LIN {X 0,Y 469.67,Z 608.611,A -85,B 0,C 180,E1 -7447.57,E2 -7447.57} C_VEL
LIN {X 0,Y 469.047,Z 617.6,A -85,B 0,C 180,E1 -7449.155,E2 -7449.155} C_VEL
LIN {X 0,Y 468.475,Z 624.989,A -85,B 0,C 180,E1 -7450.73,E2 -7450.73} C_VEL
LIN {X 0,Y 468.024,Z 631.788,A -85,B 0,C 180,E1 -7452.524,E2 -7452.524} C_VEL
LIN {X 0,Y 467.689,Z 637.041,A -85,B 0,C 180,E1 -7454.307,E2 -7454.307} C_VEL
LIN {X 0,Y 467.424,Z 640.917,A -85,B 0,C 180,E1 -7456.081,E2 -7456.081} C_VEL
LIN {X 0,Y 467.26,Z 643.569,A -85,B 0,C 180,E1 -7457.867,E2 -7457.867} C_VEL
LIN {X 0,Y 467.199,Z 644.998,A -85,B 0,C 180,E1 -7459.601,E2 -7459.601} C_VEL
LIN {X 0,Y 467.203,Z 645.333,A -85,B 0,C 180,E1 -7461.349,E2 -7461.349} C_VEL
LIN {X 0,Y 467.285,Z 644.567,A -85,B 0,C 180,E1 -7463.09,E2 -7463.09} C_VEL
LIN {X 0,Y 467.339,Z 642.693,A -85,B 0,C 180,E1 -7464.824,E2 -7464.824} C_VEL
LIN {X 0,Y 467.523,Z 639.635,A -85,B 0,C 180,E1 -7466.553,E2 -7466.553} C_VEL
LIN {X 0,Y 467.688,Z 635.408,A -85,B 0,C 180,E1 -7468.278,E2 -7468.278} C_VEL
LIN {X 0,Y 468.03,Z 629.881,A -85,B 0,C 180,E1 -7470,E2 -7470} C_VEL
LIN {X 0,Y 468.557,Z 622.901,A -85,B 0,C 180,E1 -7471.719,E2 -7471.719} C_VEL
LIN {X 0,Y 469.049,Z 615.461,A -85,B 0,C 180,E1 -7473.221,E2 -7473.221} C_VEL
LIN {X 0,Y 469.708,Z 606.525,A -85,B 0,C 180,E1 -7474.721,E2 -7474.721} C_VEL
LIN {X 0,Y 470.4,Z 597.458,A -85,B 0,C 180,E1 -7476.003,E2 -7476.003} C_VEL
LIN {X 0,Y 471.082,Z 586.721,A -85,B 0,C 180,E1 -7477.285,E2 -7477.285} C_VEL
LIN {X 0,Y 471.807,Z 574.946,A -85,B 0,C 180,E1 -7478.459,E2 -7478.459} C_VEL
LIN {X 0,Y 472.642,Z 561.989,A -85,B 0,C 180,E1 -7479.522,E2 -7479.522} C_VEL
LIN {X 0,Y 473.369,Z 547.59,A -85,B 0,C 180,E1 -7480.479,E2 -7480.479} C_VEL
LIN {X 0,Y 473.972,Z 533.272,A -85,B 0,C 180,E1 -7481.223,E2 -7481.223} C_VEL
LIN {X 0,Y 474.382,Z 517.89,A -85,B 0,C 180,E1 -7481.826,E2 -7481.826} C_VEL
LIN {X 0,Y 474.573,Z 502.138,A -85,B 0,C 180,E1 -7482.25,E2 -7482.25} C_VEL
LIN {X 0,Y 475.64,Z 391.415,A -85,B 0,C 180,E1 -7483.988,E2 -7483.988} C_VEL
LIN {X 0,Y 467.72,Z 373.635,A -85,B 0,C 180,E1 -7484.679,E2 -7484.679} C_VEL
LIN {X 0,Y 467.562,Z 372.871,A -85,B 0,C 180,E1 -7484.716,E2 -7484.716} C_VEL
LIN {X 0,Y 467.562,Z 372.866,A -85,B 0,C 180,E1 -7487.495,E2 -7487.495} C_VEL
LIN {X 0,Y 467.593,Z 372.862,A -85,B 0,C 180,E1 -7490.224,E2 -7490.224} C_VEL
LIN {X 0,Y 467.567,Z 372.868,A -85,B 0,C 180,E1 -7493.523,E2 -7493.523} C_VEL
LIN {X 0,Y 467.525,Z 372.875,A -85,B 0,C 180,E1 -7496.806,E2 -7496.806} C_VEL
LIN {X 0,Y 467.509,Z 372.863,A -85,B 0,C 180,E1 -7499.741,E2 -7499.741} C_VEL
LIN {X 0,Y 467.547,Z 372.871,A -85,B 0,C 180,E1 -7502.761,E2 -7502.761} C_VEL
LIN {X 0,Y 467.54,Z 372.867,A -85,B 0,C 180,E1 -7505.89,E2 -7505.89} C_VEL
LIN {X 0,Y 467.528,Z 372.874,A -85,B 0,C 180,E1 -7509.149,E2 -7509.149} C_VEL
LIN {X 0,Y 467.551,Z 372.871,A -85,B 0,C 180,E1 -7511.405,E2 -7511.405} C_VEL
LIN {X 0,Y 467.551,Z 372.87,A -85,B 0,C 180,E1 -7515.05,E2 -7515.05} C_VEL
LIN {X 0,Y 467.556,Z 372.866,A -85,B 0,C 180,E1 -7518.725,E2 -7518.725} C_VEL
LIN {X 0,Y 467.535,Z 372.866,A -85,B 0,C 180,E1 -7521.952,E2 -7521.952} C_VEL
LIN {X 0,Y 467.543,Z 372.873,A -85,B 0,C 180,E1 -7525.165,E2 -7525.165} C_VEL
LIN {X 0,Y 467.535,Z 372.868,A -85,B 0,C 180,E1 -7528.256,E2 -7528.256} C_VEL
LIN {X 0,Y 467.519,Z 372.873,A -85,B 0,C 180,E1 -7531.246,E2 -7531.246} C_VEL
LIN {X 0,Y 467.553,Z 372.865,A -85,B 0,C 180,E1 -7534.405,E2 -7534.405} C_VEL
LIN {X 0,Y 467.564,Z 372.864,A -85,B 0,C 180,E1 -7536.995,E2 -7536.995} C_VEL
LIN {X 0,Y 467.61,Z 372.859,A -85,B 0,C 180,E1 -7539.776,E2 -7539.776} C_VEL
LIN {X 0,Y 467.58,Z 372.86,A -85,B 0,C 180,E1 -7542.505,E2 -7542.505} C_VEL
LIN {X 0,Y 467.586,Z 372.866,A -85,B 0,C 180,E1 -7545.196,E2 -7545.196} C_VEL
LIN {X 0,Y 467.646,Z 372.839,A -85,B 0,C 180,E1 -7547.854,E2 -7547.854} C_VEL
LIN {X 0,Y 467.62,Z 372.849,A -85,B 0,C 180,E1 -7551.356,E2 -7551.356} C_VEL
LIN {X 0,Y 467.691,Z 372.851,A -85,B 0,C 180,E1 -7553.962,E2 -7553.962} C_VEL
LIN {X 0,Y 467.778,Z 372.838,A -85,B 0,C 180,E1 -7557.416,E2 -7557.416} C_VEL
LIN {X 0,Y 467.814,Z 372.835,A -85,B 0,C 180,E1 -7560,E2 -7560} C_VEL
LIN {X 0,Y 467.809,Z 372.831,A -85,B 0,C 180,E1 -7562.583,E2 -7562.583} C_VEL
LIN {X 0,Y 467.681,Z 372.851,A -85,B 0,C 180,E1 -7566.038,E2 -7566.038} C_VEL
LIN {X 0,Y 467.624,Z 372.853,A -85,B 0,C 180,E1 -7568.644,E2 -7568.644} C_VEL
LIN {X 0,Y 467.646,Z 372.855,A -85,B 0,C 180,E1 -7572.146,E2 -7572.146} C_VEL
LIN {X 0,Y 467.602,Z 372.865,A -85,B 0,C 180,E1 -7575.696,E2 -7575.696} C_VEL
LIN {X 0,Y 467.562,Z 372.861,A -85,B 0,C 180,E1 -7578.748,E2 -7578.748} C_VEL
LIN {X 0,Y 467.548,Z 372.869,A -85,B 0,C 180,E1 -7581.261,E2 -7581.261} C_VEL
LIN {X 0,Y 467.541,Z 372.872,A -85,B 0,C 180,E1 -7583.945,E2 -7583.945} C_VEL
LIN {X 0,Y 467.525,Z 372.867,A -85,B 0,C 180,E1 -7586.806,E2 -7586.806} C_VEL
LIN {X 0,Y 467.531,Z 372.874,A -85,B 0,C 180,E1 -7589.74,E2 -7589.74} C_VEL
LIN {X 0,Y 467.564,Z 372.861,A -85,B 0,C 180,E1 -7592.76,E2 -7592.76} C_VEL
LIN {X 0,Y 467.534,Z 372.877,A -85,B 0,C 180,E1 -7595.891,E2 -7595.891} C_VEL
LIN {X 0,Y 467.533,Z 372.864,A -85,B 0,C 180,E1 -7599.149,E2 -7599.149} C_VEL
LIN {X 0,Y 467.551,Z 372.87,A -85,B 0,C 180,E1 -7601.405,E2 -7601.405} C_VEL
LIN {X 0,Y 467.557,Z 372.865,A -85,B 0,C 180,E1 -7605.052,E2 -7605.052} C_VEL
LIN {X 0,Y 467.546,Z 372.859,A -85,B 0,C 180,E1 -7608.728,E2 -7608.728} C_VEL
LIN {X 0,Y 467.534,Z 372.875,A -85,B 0,C 180,E1 -7611.953,E2 -7611.953} C_VEL
LIN {X 0,Y 467.625,Z 373.006,A -85,B 0,C 180,E1 -7615.296,E2 -7615.296} C_VEL
LIN {X 0,Y 472.99,Z 393.471,A -85,B 0,C 180,E1 -7618.068,E2 -7618.068} C_VEL
LIN {X 0,Y 473.845,Z 397.012,A -85,B 0,C 180,E1 -7618.531,E2 -7618.531} C_VEL
LIN {X 0,Y 472.881,Z 418.835,A -85,B 0,C 180,E1 -7621.031,E2 -7621.031} C_VEL
LIN {X 0,Y 471.759,Z 444.502,A -85,B 0,C 180,E1 -7623.93,E2 -7623.93} C_VEL
LIN {X 0,Y 471.04,Z 462.048,A -85,B 0,C 180,E1 -7625.895,E2 -7625.895} C_VEL
LIN {X 0,Y 475.467,Z 492.83,A -85,B 0,C 180,E1 -7626.599,E2 -7626.599} C_VEL
LIN {X 0,Y 473.858,Z 631.608,A -85,B 0,C 180,E1 -7628.75,E2 -7628.75} C_VEL
LIN {X 0,Y 473.273,Z 647.666,A -85,B 0,C 180,E1 -7629.177,E2 -7629.177} C_VEL
LIN {X 0,Y 472.573,Z 661.612,A -85,B 0,C 180,E1 -7629.705,E2 -7629.705} C_VEL
LIN {X 0,Y 471.782,Z 675.9,A -85,B 0,C 180,E1 -7630.417,E2 -7630.417} C_VEL
LIN {X 0,Y 470.956,Z 689.732,A -85,B 0,C 180,E1 -7631.286,E2 -7631.286} C_VEL
LIN {X 0,Y 470.13,Z 702.495,A -85,B 0,C 180,E1 -7632.267,E2 -7632.267} C_VEL
LIN {X 0,Y 469.317,Z 715.487,A -85,B 0,C 180,E1 -7633.47,E2 -7633.47} C_VEL
LIN {X 0,Y 468.57,Z 727.313,A -85,B 0,C 180,E1 -7634.783,E2 -7634.783} C_VEL
LIN {X 0,Y 468.028,Z 737.298,A -85,B 0,C 180,E1 -7636.098,E2 -7636.098} C_VEL
LIN {X 0,Y 467.584,Z 746.096,A -85,B 0,C 180,E1 -7637.456,E2 -7637.456} C_VEL
LIN {X 0,Y 467.298,Z 754.281,A -85,B 0,C 180,E1 -7638.945,E2 -7638.945} C_VEL
LIN {X 0,Y 467.041,Z 761.256,A -85,B 0,C 180,E1 -7640.472,E2 -7640.472} C_VEL
LIN {X 0,Y 466.972,Z 767.735,A -85,B 0,C 180,E1 -7642.215,E2 -7642.215} C_VEL
LIN {X 0,Y 466.958,Z 772.754,A -85,B 0,C 180,E1 -7643.952,E2 -7643.952} C_VEL
LIN {X 0,Y 467.019,Z 776.441,A -85,B 0,C 180,E1 -7645.685,E2 -7645.685} C_VEL
LIN {X 0,Y 466.958,Z 778.848,A -85,B 0,C 180,E1 -7647.412,E2 -7647.412} C_VEL
LIN {X 0,Y 467.025,Z 780.065,A -85,B 0,C 180,E1 -7649.137,E2 -7649.137} C_VEL
LIN {X 0,Y 467.026,Z 780.047,A -85,B 0,C 180,E1 -7650.862,E2 -7650.862} C_VEL
LIN {X 0,Y 466.964,Z 778.797,A -85,B 0,C 180,E1 -7652.587,E2 -7652.587} C_VEL
LIN {X 0,Y 467.04,Z 776.363,A -85,B 0,C 180,E1 -7654.315,E2 -7654.315} C_VEL
LIN {X 0,Y 466.966,Z 772.648,A -85,B 0,C 180,E1 -7656.047,E2 -7656.047} C_VEL
LIN {X 0,Y 466.981,Z 767.598,A -85,B 0,C 180,E1 -7657.784,E2 -7657.784} C_VEL
LIN {X 0,Y 467.071,Z 761.078,A -85,B 0,C 180,E1 -7659.527,E2 -7659.527} C_VEL
LIN {X 0,Y 467.296,Z 754.064,A -85,B 0,C 180,E1 -7661.055,E2 -7661.055} C_VEL
LIN {X 0,Y 467.591,Z 745.859,A -85,B 0,C 180,E1 -7662.543,E2 -7662.543} C_VEL
LIN {X 0,Y 468.026,Z 737.049,A -85,B 0,C 180,E1 -7663.901,E2 -7663.901} C_VEL
LIN {X 0,Y 468.578,Z 727.074,A -85,B 0,C 180,E1 -7665.216,E2 -7665.216} C_VEL
LIN {X 0,Y 469.304,Z 714.794,A -85,B 0,C 180,E1 -7666.58,E2 -7666.58} C_VEL
LIN {X 0,Y 470.115,Z 702.374,A -85,B 0,C 180,E1 -7667.733,E2 -7667.733} C_VEL
LIN {X 0,Y 470.899,Z 689.72,A -85,B 0,C 180,E1 -7668.715,E2 -7668.715} C_VEL
LIN {X 0,Y 471.784,Z 676.095,A -85,B 0,C 180,E1 -7669.582,E2 -7669.582} C_VEL
LIN {X 0,Y 472.598,Z 662.069,A -85,B 0,C 180,E1 -7670.293,E2 -7670.293} C_VEL
LIN {X 0,Y 473.391,Z 646.192,A -85,B 0,C 180,E1 -7670.901,E2 -7670.901} C_VEL
LIN {X 0,Y 473.955,Z 630.96,A -85,B 0,C 180,E1 -7671.302,E2 -7671.302} C_VEL
LIN {X 0,Y 475.444,Z 512.492,A -85,B 0,C 180,E1 -7673.158,E2 -7673.158} C_VEL
LIN {X 0,Y 475.512,Z 491.468,A -85,B 0,C 180,E1 -7673.495,E2 -7673.495} C_VEL
LIN {X 0,Y 471.127,Z 461.112,A -85,B 0,C 180,E1 -7674.248,E2 -7674.248} C_VEL
LIN {X 0,Y 472.502,Z 431.974,A -85,B 0,C 180,E1 -7677.577,E2 -7677.577} C_VEL
LIN {X 0,Y 473.976,Z 403.693,A -85,B 0,C 180,E1 -7680.877,E2 -7680.877} C_VEL
LIN {X 0,Y 474.148,Z 396.929,A -85,B 0,C 180,E1 -7681.691,E2 -7681.691} C_VEL
LIN {X 0,Y 469.857,Z 380.816,A -85,B 0,C 180,E1 -7683.982,E2 -7683.982} C_VEL
LIN {X 0,Y 467.577,Z 372.866,A -85,B 0,C 180,E1 -7685.192,E2 -7685.192} C_VEL
LIN {X 0,Y 467.533,Z 372.874,A -85,B 0,C 180,E1 -7688.587,E2 -7688.587} C_VEL
LIN {X 0,Y 467.552,Z 372.866,A -85,B 0,C 180,E1 -7691.404,E2 -7691.404} C_VEL
LIN {X 0,Y 467.553,Z 372.858,A -85,B 0,C 180,E1 -7694.947,E2 -7694.947} C_VEL
LIN {X 0,Y 467.547,Z 372.868,A -85,B 0,C 180,E1 -7698.594,E2 -7698.594} C_VEL
LIN {X 0,Y 467.529,Z 372.866,A -85,B 0,C 180,E1 -7701.412,E2 -7701.412} C_VEL
LIN {X 0,Y 467.537,Z 372.872,A -85,B 0,C 180,E1 -7704.262,E2 -7704.262} C_VEL
LIN {X 0,Y 467.559,Z 372.866,A -85,B 0,C 180,E1 -7707.323,E2 -7707.323} C_VEL
LIN {X 0,Y 467.536,Z 372.873,A -85,B 0,C 180,E1 -7710.672,E2 -7710.672} C_VEL
LIN {X 0,Y 467.52,Z 372.871,A -85,B 0,C 180,E1 -7713.194,E2 -7713.194} C_VEL
LIN {X 0,Y 467.536,Z 372.871,A -85,B 0,C 180,E1 -7716.055,E2 -7716.055} C_VEL
LIN {X 0,Y 467.571,Z 372.863,A -85,B 0,C 180,E1 -7719.775,E2 -7719.775} C_VEL
LIN {X 0,Y 467.542,Z 372.871,A -85,B 0,C 180,E1 -7722.504,E2 -7722.504} C_VEL
LIN {X 0,Y 467.571,Z 372.864,A -85,B 0,C 180,E1 -7725.196,E2 -7725.196} C_VEL
LIN {X 0,Y 467.641,Z 372.857,A -85,B 0,C 180,E1 -7727.854,E2 -7727.854} C_VEL
LIN {X 0,Y 467.619,Z 372.858,A -85,B 0,C 180,E1 -7731.356,E2 -7731.356} C_VEL
LIN {X 0,Y 467.677,Z 372.848,A -85,B 0,C 180,E1 -7733.962,E2 -7733.962} C_VEL
LIN {X 0,Y 467.805,Z 372.83,A -85,B 0,C 180,E1 -7737.417,E2 -7737.417} C_VEL
LIN {X 0,Y 467.831,Z 372.833,A -85,B 0,C 180,E1 -7740,E2 -7740} C_VEL
LIN {X 0,Y 467.803,Z 372.84,A -85,B 0,C 180,E1 -7742.583,E2 -7742.583} C_VEL
LIN {X 0,Y 467.706,Z 372.84,A -85,B 0,C 180,E1 -7746.038,E2 -7746.038} C_VEL
LIN {X 0,Y 467.646,Z 372.849,A -85,B 0,C 180,E1 -7748.644,E2 -7748.644} C_VEL
LIN {X 0,Y 467.641,Z 372.856,A -85,B 0,C 180,E1 -7752.146,E2 -7752.146} C_VEL
LIN {X 0,Y 467.636,Z 372.85,A -85,B 0,C 180,E1 -7755.885,E2 -7755.885} C_VEL
LIN {X 0,Y 467.609,Z 372.854,A -85,B 0,C 180,E1 -7759.309,E2 -7759.309} C_VEL
LIN {X 0,Y 467.518,Z 372.864,A -85,B 0,C 180,E1 -7762.075,E2 -7762.075} C_VEL
LIN {X 0,Y 467.543,Z 372.87,A -85,B 0,C 180,E1 -7764.891,E2 -7764.891} C_VEL
LIN {X 0,Y 467.535,Z 372.865,A -85,B 0,C 180,E1 -7767.775,E2 -7767.775} C_VEL
LIN {X 0,Y 467.54,Z 372.866,A -85,B 0,C 180,E1 -7771.042,E2 -7771.042} C_VEL
LIN {X 0,Y 467.567,Z 372.867,A -85,B 0,C 180,E1 -7774.241,E2 -7774.241} C_VEL
LIN {X 0,Y 467.538,Z 372.869,A -85,B 0,C 180,E1 -7777.187,E2 -7777.187} C_VEL
LIN {X 0,Y 467.549,Z 372.866,A -85,B 0,C 180,E1 -7780.268,E2 -7780.268} C_VEL
LIN {X 0,Y 467.539,Z 372.863,A -85,B 0,C 180,E1 -7783.747,E2 -7783.747} C_VEL
LIN {X 0,Y 467.54,Z 372.869,A -85,B 0,C 180,E1 -7786.256,E2 -7786.256} C_VEL
LIN {X 0,Y 467.553,Z 372.866,A -85,B 0,C 180,E1 -7789.735,E2 -7789.735} C_VEL
LIN {X 0,Y 467.538,Z 372.871,A -85,B 0,C 180,E1 -7792.816,E2 -7792.816} C_VEL
LIN {X 0,Y 467.572,Z 372.868,A -85,B 0,C 180,E1 -7795.761,E2 -7795.761} C_VEL
LIN {X 0,Y 467.592,Z 372.908,A -85,B 0,C 180,E1 -7797.131,E2 -7797.131} C_VEL
LIN {X 0,Y 468.547,Z 375.634,A -85,B 0,C 180,E1 -7797.236,E2 -7797.236} C_VEL
LIN {X 0,Y 476.262,Z 391.882,A -85,B 0,C 180,E1 -7797.966,E2 -7797.966} C_VEL
LIN {X 0,Y 475.026,Z 501.799,A -85,B 0,C 180,E1 -7799.71,E2 -7799.71} C_VEL
LIN {X 0,Y 475.018,Z 504.372,A -85,B 0,C 180,E1 -7799.763,E2 -7799.763} C_VEL
LIN {X 0,Y 474.664,Z 508.241,A -85,B 0,C 180,E1 -7799.84,E2 -7799.84} C_VEL
LIN {X 0,Y 472.596,Z 515.855,A -85,B 0,C 180,E1 -7799.943,E2 -7799.943} C_VEL
LIN {X 0,Y 468.602,Z 527.997,A -85,B 0,C 180,E1 -7800.171,E2 -7800.171} C_VEL
LIN {X 0,Y 467.913,Z 532.637,A -85,B 0,C 180,E1 -7800.343,E2 -7800.343} C_VEL
LIN {X 0,Y 467.847,Z 534.491,A -85,B 0,C 180,E1 -7800.424,E2 -7800.424} C_VEL
LIN {X 0,Y 467.113,Z 549.49,A -85,B 0,C 180,E1 -7801.22,E2 -7801.22} C_VEL
LIN {X 0,Y 466.385,Z 563.17,A -85,B 0,C 180,E1 -7802.152,E2 -7802.152} C_VEL
LIN {X 0,Y 465.508,Z 576.883,A -85,B 0,C 180,E1 -7803.312,E2 -7803.312} C_VEL
LIN {X 0,Y 464.664,Z 588.188,A -85,B 0,C 180,E1 -7804.466,E2 -7804.466} C_VEL
LIN {X 0,Y 463.782,Z 599.464,A -85,B 0,C 180,E1 -7805.85,E2 -7805.85} C_VEL
LIN {X 0,Y 462.959,Z 608.86,A -85,B 0,C 180,E1 -7807.227,E2 -7807.227} C_VEL
LIN {X 0,Y 462.247,Z 617.984,A -85,B 0,C 180,E1 -7808.833,E2 -7808.833} C_VEL
LIN {X 0,Y 461.623,Z 625.471,A -85,B 0,C 180,E1 -7810.432,E2 -7810.432} C_VEL
LIN {X 0,Y 461.126,Z 632.379,A -85,B 0,C 180,E1 -7812.254,E2 -7812.254} C_VEL
LIN {X 0,Y 460.729,Z 637.73,A -85,B 0,C 180,E1 -7814.064,E2 -7814.064} C_VEL
LIN {X 0,Y 460.459,Z 641.695,A -85,B 0,C 180,E1 -7815.866,E2 -7815.866} C_VEL
LIN {X 0,Y 460.26,Z 644.531,A -85,B 0,C 180,E1 -7817.758,E2 -7817.758} C_VEL
LIN {X 0,Y 460.18,Z 645.952,A -85,B 0,C 180,E1 -7819.441,E2 -7819.441} C_VEL
LIN {X 0,Y 460.192,Z 646.37,A -85,B 0,C 180,E1 -7821.216,E2 -7821.216} C_VEL
LIN {X 0,Y 460.269,Z 645.681,A -85,B 0,C 180,E1 -7822.984,E2 -7822.984} C_VEL
LIN {X 0,Y 460.33,Z 643.853,A -85,B 0,C 180,E1 -7824.745,E2 -7824.745} C_VEL
LIN {X 0,Y 460.485,Z 640.888,A -85,B 0,C 180,E1 -7826.5,E2 -7826.5} C_VEL
LIN {X 0,Y 460.692,Z 636.744,A -85,B 0,C 180,E1 -7828.252,E2 -7828.252} C_VEL
LIN {X 0,Y 461.044,Z 631.311,A -85,B 0,C 180,E1 -7830,E2 -7830} C_VEL
LIN {X 0,Y 461.586,Z 624.434,A -85,B 0,C 180,E1 -7831.745,E2 -7831.745} C_VEL
LIN {X 0,Y 462.11,Z 617.103,A -85,B 0,C 180,E1 -7833.27,E2 -7833.27} C_VEL
LIN {X 0,Y 462.788,Z 608.296,A -85,B 0,C 180,E1 -7834.791,E2 -7834.791} C_VEL
LIN {X 0,Y 463.52,Z 599.322,A -85,B 0,C 180,E1 -7836.093,E2 -7836.093} C_VEL
LIN {X 0,Y 464.225,Z 588.721,A -85,B 0,C 180,E1 -7837.394,E2 -7837.394} C_VEL
LIN {X 0,Y 464.964,Z 577.141,A -85,B 0,C 180,E1 -7838.584,E2 -7838.584} C_VEL
LIN {X 0,Y 465.853,Z 564.424,A -85,B 0,C 180,E1 -7839.662,E2 -7839.662} C_VEL
LIN {X 0,Y 466.513,Z 552.091,A -85,B 0,C 180,E1 -7840.525,E2 -7840.525} C_VEL
LIN {X 0,Y 467.153,Z 538.751,A -85,B 0,C 180,E1 -7841.278,E2 -7841.278} C_VEL
LIN {X 0,Y 467.643,Z 524.035,A -85,B 0,C 180,E1 -7841.923,E2 -7841.923} C_VEL
LIN {X 0,Y 467.888,Z 509.404,A -85,B 0,C 180,E1 -7842.39,E2 -7842.39} C_VEL
LIN {X 0,Y 468.007,Z 493.494,A -85,B 0,C 180,E1 -7842.714,E2 -7842.714} C_VEL
LIN {X 0,Y 469.054,Z 393.357,A -85,B 0,C 180,E1 -7844.288,E2 -7844.288} C_VEL
LIN {X 0,Y 460.595,Z 374.2,A -85,B 0,C 180,E1 -7845.043,E2 -7845.043} C_VEL
LIN {X 0,Y 460.516,Z 373.749,A -85,B 0,C 180,E1 -7845.093,E2 -7845.093} C_VEL
LIN {X 0,Y 460.516,Z 373.744,A -85,B 0,C 180,E1 -7847.771,E2 -7847.771} C_VEL
LIN {X 0,Y 460.527,Z 373.744,A -85,B 0,C 180,E1 -7850.548,E2 -7850.548} C_VEL
LIN {X 0,Y 460.504,Z 373.747,A -85,B 0,C 180,E1 -7853.695,E2 -7853.695} C_VEL
LIN {X 0,Y 460.479,Z 373.749,A -85,B 0,C 180,E1 -7856.27,E2 -7856.27} C_VEL
LIN {X 0,Y 460.497,Z 373.741,A -85,B 0,C 180,E1 -7859.233,E2 -7859.233} C_VEL
LIN {X 0,Y 460.496,Z 373.746,A -85,B 0,C 180,E1 -7862.287,E2 -7862.287} C_VEL
LIN {X 0,Y 460.496,Z 373.749,A -85,B 0,C 180,E1 -7865.446,E2 -7865.446} C_VEL
LIN {X 0,Y 460.481,Z 373.752,A -85,B 0,C 180,E1 -7868.887,E2 -7868.887} C_VEL
LIN {X 0,Y 460.496,Z 373.748,A -85,B 0,C 180,E1 -7871.597,E2 -7871.597} C_VEL
LIN {X 0,Y 460.494,Z 373.744,A -85,B 0,C 180,E1 -7874.59,E2 -7874.59} C_VEL
LIN {X 0,Y 460.469,Z 373.748,A -85,B 0,C 180,E1 -7877.812,E2 -7877.812} C_VEL
LIN {X 0,Y 460.504,Z 373.744,A -85,B 0,C 180,E1 -7880.134,E2 -7880.134} C_VEL
LIN {X 0,Y 460.458,Z 373.756,A -85,B 0,C 180,E1 -7883.469,E2 -7883.469} C_VEL
LIN {X 0,Y 460.494,Z 373.742,A -85,B 0,C 180,E1 -7886.672,E2 -7886.672} C_VEL
LIN {X 0,Y 460.472,Z 373.748,A -85,B 0,C 180,E1 -7889.757,E2 -7889.757} C_VEL
LIN {X 0,Y 460.476,Z 373.748,A -85,B 0,C 180,E1 -7892.75,E2 -7892.75} C_VEL
LIN {X 0,Y 460.504,Z 373.743,A -85,B 0,C 180,E1 -7895.665,E2 -7895.665} C_VEL
LIN {X 0,Y 460.514,Z 373.743,A -85,B 0,C 180,E1 -7898.578,E2 -7898.578} C_VEL
LIN {X 0,Y 460.574,Z 373.736,A -85,B 0,C 180,E1 -7901.31,E2 -7901.31} C_VEL
LIN {X 0,Y 460.578,Z 373.735,A -85,B 0,C 180,E1 -7904.058,E2 -7904.058} C_VEL
LIN {X 0,Y 460.6,Z 373.718,A -85,B 0,C 180,E1 -7907.665,E2 -7907.665} C_VEL
LIN {X 0,Y 460.576,Z 373.724,A -85,B 0,C 180,E1 -7911.223,E2 -7911.223} C_VEL
LIN {X 0,Y 460.657,Z 373.728,A -85,B 0,C 180,E1 -7913.869,E2 -7913.869} C_VEL
LIN {X 0,Y 460.725,Z 373.716,A -85,B 0,C 180,E1 -7917.377,E2 -7917.377} C_VEL
LIN {X 0,Y 460.764,Z 373.713,A -85,B 0,C 180,E1 -7920,E2 -7920} C_VEL
LIN {X 0,Y 460.753,Z 373.71,A -85,B 0,C 180,E1 -7922.623,E2 -7922.623} C_VEL
LIN {X 0,Y 460.648,Z 373.727,A -85,B 0,C 180,E1 -7926.131,E2 -7926.131} C_VEL
LIN {X 0,Y 460.579,Z 373.73,A -85,B 0,C 180,E1 -7928.777,E2 -7928.777} C_VEL
LIN {X 0,Y 460.599,Z 373.732,A -85,B 0,C 180,E1 -7932.334,E2 -7932.334} C_VEL
LIN {X 0,Y 460.548,Z 373.743,A -85,B 0,C 180,E1 -7935.978,E2 -7935.978} C_VEL
LIN {X 0,Y 460.52,Z 373.738,A -85,B 0,C 180,E1 -7938.886,E2 -7938.886} C_VEL
LIN {X 0,Y 460.499,Z 373.75,A -85,B 0,C 180,E1 -7941.486,E2 -7941.486} C_VEL
LIN {X 0,Y 460.506,Z 373.745,A -85,B 0,C 180,E1 -7944.334,E2 -7944.334} C_VEL
LIN {X 0,Y 460.481,Z 373.747,A -85,B 0,C 180,E1 -7947.249,E2 -7947.249} C_VEL
LIN {X 0,Y 460.492,Z 373.749,A -85,B 0,C 180,E1 -7950.241,E2 -7950.241} C_VEL
LIN {X 0,Y 460.507,Z 373.743,A -85,B 0,C 180,E1 -7953.326,E2 -7953.326} C_VEL
LIN {X 0,Y 460.451,Z 373.753,A -85,B 0,C 180,E1 -7956.532,E2 -7956.532} C_VEL
LIN {X 0,Y 460.501,Z 373.749,A -85,B 0,C 180,E1 -7959.865,E2 -7959.865} C_VEL
LIN {X 0,Y 460.452,Z 373.748,A -85,B 0,C 180,E1 -7962.893,E2 -7962.893} C_VEL
LIN {X 0,Y 460.497,Z 373.747,A -85,B 0,C 180,E1 -7965.832,E2 -7965.832} C_VEL
LIN {X 0,Y 460.495,Z 373.736,A -85,B 0,C 180,E1 -7968.986,E2 -7968.986} C_VEL
LIN {X 0,Y 460.477,Z 373.753,A -85,B 0,C 180,E1 -7972.375,E2 -7972.375} C_VEL
LIN {X 0,Y 460.537,Z 373.758,A -85,B 0,C 180,E1 -7974.956,E2 -7974.956} C_VEL
LIN {X 0,Y 465.718,Z 393.481,A -85,B 0,C 180,E1 -7977.68,E2 -7977.68} C_VEL
LIN {X 0,Y 467.055,Z 399.5,A -85,B 0,C 180,E1 -7978.474,E2 -7978.474} C_VEL
LIN {X 0,Y 465.927,Z 422.481,A -85,B 0,C 180,E1 -7981.14,E2 -7981.14} C_VEL
LIN {X 0,Y 464.771,Z 447.384,A -85,B 0,C 180,E1 -7983.991,E2 -7983.991} C_VEL
LIN {X 0,Y 464.175,Z 461.003,A -85,B 0,C 180,E1 -7985.539,E2 -7985.539} C_VEL
LIN {X 0,Y 468.822,Z 493.715,A -85,B 0,C 180,E1 -7986.299,E2 -7986.299} C_VEL
LIN {X 0,Y 467.199,Z 629.756,A -85,B 0,C 180,E1 -7988.432,E2 -7988.432} C_VEL
LIN {X 0,Y 466.625,Z 645.698,A -85,B 0,C 180,E1 -7988.85,E2 -7988.85} C_VEL
LIN {X 0,Y 465.829,Z 660.502,A -85,B 0,C 180,E1 -7989.411,E2 -7989.411} C_VEL
LIN {X 0,Y 465.022,Z 674.608,A -85,B 0,C 180,E1 -7990.12,E2 -7990.12} C_VEL
LIN {X 0,Y 464.097,Z 688.498,A -85,B 0,C 180,E1 -7990.999,E2 -7990.999} C_VEL
LIN {X 0,Y 463.256,Z 701.315,A -85,B 0,C 180,E1 -7991.995,E2 -7991.995} C_VEL
LIN {X 0,Y 462.473,Z 713.255,A -85,B 0,C 180,E1 -7993.104,E2 -7993.104} C_VEL
LIN {X 0,Y 461.714,Z 724.368,A -85,B 0,C 180,E1 -7994.325,E2 -7994.325} C_VEL
LIN {X 0,Y 461.078,Z 734.675,A -85,B 0,C 180,E1 -7995.659,E2 -7995.659} C_VEL
LIN {X 0,Y 460.573,Z 744.783,A -85,B 0,C 180,E1 -7997.217,E2 -7997.217} C_VEL
LIN {X 0,Y 460.226,Z 753.234,A -85,B 0,C 180,E1 -7998.773,E2 -7998.773} C_VEL
LIN {X 0,Y 459.97,Z 760.223,A -85,B 0,C 180,E1 -8000.324,E2 -8000.324} C_VEL
LIN {X 0,Y 459.93,Z 766.715,A -85,B 0,C 180,E1 -8002.095,E2 -8002.095} C_VEL
LIN {X 0,Y 459.907,Z 771.737,A -85,B 0,C 180,E1 -8003.859,E2 -8003.859} C_VEL
LIN {X 0,Y 459.974,Z 775.427,A -85,B 0,C 180,E1 -8005.618,E2 -8005.618} C_VEL
LIN {X 0,Y 459.92,Z 777.835,A -85,B 0,C 180,E1 -8007.372,E2 -8007.372} C_VEL
LIN {X 0,Y 460.011,Z 779.054,A -85,B 0,C 180,E1 -8009.124,E2 -8009.124} C_VEL
LIN {X 0,Y 460.011,Z 779.033,A -85,B 0,C 180,E1 -8010.875,E2 -8010.875} C_VEL
LIN {X 0,Y 459.926,Z 777.776,A -85,B 0,C 180,E1 -8012.627,E2 -8012.627} C_VEL
LIN {X 0,Y 459.996,Z 775.336,A -85,B 0,C 180,E1 -8014.381,E2 -8014.381} C_VEL
LIN {X 0,Y 459.918,Z 771.617,A -85,B 0,C 180,E1 -8016.14,E2 -8016.14} C_VEL
LIN {X 0,Y 459.936,Z 766.563,A -85,B 0,C 180,E1 -8017.904,E2 -8017.904} C_VEL
LIN {X 0,Y 459.991,Z 760.039,A -85,B 0,C 180,E1 -8019.675,E2 -8019.675} C_VEL
LIN {X 0,Y 460.22,Z 753.027,A -85,B 0,C 180,E1 -8021.227,E2 -8021.227} C_VEL
LIN {X 0,Y 460.574,Z 744.583,A -85,B 0,C 180,E1 -8022.782,E2 -8022.782} C_VEL
LIN {X 0,Y 461.098,Z 734.509,A -85,B 0,C 180,E1 -8024.34,E2 -8024.34} C_VEL
LIN {X 0,Y 461.707,Z 724.259,A -85,B 0,C 180,E1 -8025.675,E2 -8025.675} C_VEL
LIN {X 0,Y 462.531,Z 712.158,A -85,B 0,C 180,E1 -8027.007,E2 -8027.007} C_VEL
LIN {X 0,Y 463.445,Z 698.843,A -85,B 0,C 180,E1 -8028.225,E2 -8028.225} C_VEL
LIN {X 0,Y 464.292,Z 685.673,A -85,B 0,C 180,E1 -8029.221,E2 -8029.221} C_VEL
LIN {X 0,Y 465.283,Z 671.331,A -85,B 0,C 180,E1 -8030.098,E2 -8030.098} C_VEL
LIN {X 0,Y 466.169,Z 656.601,A -85,B 0,C 180,E1 -8030.803,E2 -8030.803} C_VEL
LIN {X 0,Y 466.958,Z 641.178,A -85,B 0,C 180,E1 -8031.347,E2 -8031.347} C_VEL
LIN {X 0,Y 467.494,Z 625.052,A -85,B 0,C 180,E1 -8031.727,E2 -8031.727} C_VEL
LIN {X 0,Y 469.125,Z 493.023,A -85,B 0,C 180,E1 -8033.815,E2 -8033.815} C_VEL
LIN {X 0,Y 464.332,Z 459.981,A -85,B 0,C 180,E1 -8034.657,E2 -8034.657} C_VEL
LIN {X 0,Y 465.808,Z 431.181,A -85,B 0,C 180,E1 -8038.008,E2 -8038.008} C_VEL
LIN {X 0,Y 467.299,Z 404.913,A -85,B 0,C 180,E1 -8041.126,E2 -8041.126} C_VEL
LIN {X 0,Y 467.523,Z 399.827,A -85,B 0,C 180,E1 -8041.743,E2 -8041.743} C_VEL
LIN {X 0,Y 464.244,Z 386.595,A -85,B 0,C 180,E1 -8043.631,E2 -8043.631} C_VEL
LIN {X 0,Y 460.521,Z 373.743,A -85,B 0,C 180,E1 -8045.601,E2 -8045.601} C_VEL
LIN {X 0,Y 460.483,Z 373.751,A -85,B 0,C 180,E1 -8048.888,E2 -8048.888} C_VEL
LIN {X 0,Y 460.496,Z 373.747,A -85,B 0,C 180,E1 -8051.598,E2 -8051.598} C_VEL
LIN {X 0,Y 460.501,Z 373.739,A -85,B 0,C 180,E1 -8054.589,E2 -8054.589} C_VEL
LIN {X 0,Y 460.463,Z 373.752,A -85,B 0,C 180,E1 -8057.812,E2 -8057.812} C_VEL
LIN {X 0,Y 460.499,Z 373.751,A -85,B 0,C 180,E1 -8060.134,E2 -8060.134} C_VEL
LIN {X 0,Y 460.447,Z 373.751,A -85,B 0,C 180,E1 -8063.468,E2 -8063.468} C_VEL
LIN {X 0,Y 460.503,Z 373.747,A -85,B 0,C 180,E1 -8066.673,E2 -8066.673} C_VEL
LIN {X 0,Y 460.488,Z 373.746,A -85,B 0,C 180,E1 -8069.759,E2 -8069.759} C_VEL
LIN {X 0,Y 460.477,Z 373.751,A -85,B 0,C 180,E1 -8072.75,E2 -8072.75} C_VEL
LIN {X 0,Y 460.501,Z 373.745,A -85,B 0,C 180,E1 -8075.666,E2 -8075.666} C_VEL
LIN {X 0,Y 460.499,Z 373.747,A -85,B 0,C 180,E1 -8078.581,E2 -8078.581} C_VEL
LIN {X 0,Y 460.515,Z 373.744,A -85,B 0,C 180,E1 -8081.308,E2 -8081.308} C_VEL
LIN {X 0,Y 460.552,Z 373.741,A -85,B 0,C 180,E1 -8084.057,E2 -8084.057} C_VEL
LIN {X 0,Y 460.594,Z 373.733,A -85,B 0,C 180,E1 -8087.666,E2 -8087.666} C_VEL
LIN {X 0,Y 460.574,Z 373.736,A -85,B 0,C 180,E1 -8091.223,E2 -8091.223} C_VEL
LIN {X 0,Y 460.644,Z 373.723,A -85,B 0,C 180,E1 -8093.869,E2 -8093.869} C_VEL
LIN {X 0,Y 460.75,Z 373.709,A -85,B 0,C 180,E1 -8097.377,E2 -8097.377} C_VEL
LIN {X 0,Y 460.78,Z 373.711,A -85,B 0,C 180,E1 -8100,E2 -8100} C_VEL
LIN {X 0,Y 460.747,Z 373.719,A -85,B 0,C 180,E1 -8102.623,E2 -8102.623} C_VEL
LIN {X 0,Y 460.672,Z 373.715,A -85,B 0,C 180,E1 -8106.131,E2 -8106.131} C_VEL
LIN {X 0,Y 460.594,Z 373.729,A -85,B 0,C 180,E1 -8108.777,E2 -8108.777} C_VEL
LIN {X 0,Y 460.595,Z 373.735,A -85,B 0,C 180,E1 -8112.335,E2 -8112.335} C_VEL
LIN {X 0,Y 460.588,Z 373.728,A -85,B 0,C 180,E1 -8115.998,E2 -8115.998} C_VEL
LIN {X 0,Y 460.555,Z 373.731,A -85,B 0,C 180,E1 -8119.616,E2 -8119.616} C_VEL
LIN {X 0,Y 460.495,Z 373.741,A -85,B 0,C 180,E1 -8122.43,E2 -8122.43} C_VEL
LIN {X 0,Y 460.521,Z 373.737,A -85,B 0,C 180,E1 -8125.793,E2 -8125.793} C_VEL
LIN {X 0,Y 460.511,Z 373.748,A -85,B 0,C 180,E1 -8129.233,E2 -8129.233} C_VEL
LIN {X 0,Y 460.515,Z 373.736,A -85,B 0,C 180,E1 -8132.286,E2 -8132.286} C_VEL
LIN {X 0,Y 460.499,Z 373.745,A -85,B 0,C 180,E1 -8135.447,E2 -8135.447} C_VEL
LIN {X 0,Y 460.521,Z 373.75,A -85,B 0,C 180,E1 -8138.896,E2 -8138.896} C_VEL
LIN {X 0,Y 460.471,Z 373.749,A -85,B 0,C 180,E1 -8142.188,E2 -8142.188} C_VEL
LIN {X 0,Y 460.505,Z 373.748,A -85,B 0,C 180,E1 -8145.412,E2 -8145.412} C_VEL
LIN {X 0,Y 460.513,Z 373.747,A -85,B 0,C 180,E1 -8148.988,E2 -8148.988} C_VEL
LIN {X 0,Y 460.509,Z 373.747,A -85,B 0,C 180,E1 -8151.267,E2 -8151.267} C_VEL
LIN {X 0,Y 460.502,Z 373.745,A -85,B 0,C 180,E1 -8154.555,E2 -8154.555} C_VEL
LIN {X 0,Y 460.527,Z 373.746,A -85,B 0,C 180,E1 -8156.676,E2 -8156.676} C_VEL
LIN {X 0,Y 461.674,Z 376.815,A -85,B 0,C 180,E1 -8156.823,E2 -8156.823} C_VEL
LIN {X 0,Y 469.854,Z 393.695,A -85,B 0,C 180,E1 -8157.618,E2 -8157.618} C_VEL
LIN {X 0,Y 468.547,Z 502.603,A -85,B 0,C 180,E1 -8159.37,E2 -8159.37} C_VEL
LIN {X 0,Y 468.329,Z 517.419,A -85,B 0,C 180,E1 -8159.759,E2 -8159.759} C_VEL
LIN {X 0,Y 467.91,Z 531.431,A -85,B 0,C 180,E1 -8160.288,E2 -8160.288} C_VEL
LIN {X 0,Y 467.847,Z 534.491,A -85,B 0,C 180,E1 -8160.424,E2 -8160.424} C_VEL
LIN {X 0,Y 467.117,Z 540.043,A -85,B 0,C 180,E1 -8160.657,E2 -8160.657} C_VEL
LIN {X 0,Y 463.965,Z 549.047,A -85,B 0,C 180,E1 -8161.002,E2 -8161.002} C_VEL
LIN {X 0,Y 460.736,Z 557.83,A -85,B 0,C 180,E1 -8161.413,E2 -8161.413} C_VEL
LIN {X 0,Y 459.863,Z 562.966,A -85,B 0,C 180,E1 -8161.753,E2 -8161.753} C_VEL
LIN {X 0,Y 459.064,Z 575.115,A -85,B 0,C 180,E1 -8162.763,E2 -8162.763} C_VEL
LIN {X 0,Y 458.159,Z 587.034,A -85,B 0,C 180,E1 -8163.955,E2 -8163.955} C_VEL
LIN {X 0,Y 457.213,Z 598.568,A -85,B 0,C 180,E1 -8165.344,E2 -8165.344} C_VEL
LIN {X 0,Y 456.255,Z 609.112,A -85,B 0,C 180,E1 -8166.873,E2 -8166.873} C_VEL
LIN {X 0,Y 455.472,Z 618.368,A -85,B 0,C 180,E1 -8168.503,E2 -8168.503} C_VEL
LIN {X 0,Y 454.767,Z 625.971,A -85,B 0,C 180,E1 -8170.125,E2 -8170.125} C_VEL
LIN {X 0,Y 454.223,Z 632.982,A -85,B 0,C 180,E1 -8171.975,E2 -8171.975} C_VEL
LIN {X 0,Y 453.814,Z 638.427,A -85,B 0,C 180,E1 -8173.815,E2 -8173.815} C_VEL
LIN {X 0,Y 453.483,Z 642.484,A -85,B 0,C 180,E1 -8175.644,E2 -8175.644} C_VEL
LIN {X 0,Y 453.278,Z 645.485,A -85,B 0,C 180,E1 -8177.637,E2 -8177.637} C_VEL
LIN {X 0,Y 453.167,Z 646.909,A -85,B 0,C 180,E1 -8179.275,E2 -8179.275} C_VEL
LIN {X 0,Y 453.191,Z 647.406,A -85,B 0,C 180,E1 -8181.079,E2 -8181.079} C_VEL
LIN {X 0,Y 453.25,Z 646.739,A -85,B 0,C 180,E1 -8182.921,E2 -8182.921} C_VEL
LIN {X 0,Y 453.321,Z 645.008,A -85,B 0,C 180,E1 -8184.663,E2 -8184.663} C_VEL
LIN {X 0,Y 453.449,Z 642.133,A -85,B 0,C 180,E1 -8186.446,E2 -8186.446} C_VEL
LIN {X 0,Y 453.695,Z 638.07,A -85,B 0,C 180,E1 -8188.225,E2 -8188.225} C_VEL
LIN {X 0,Y 454.053,Z 632.731,A -85,B 0,C 180,E1 -8190,E2 -8190} C_VEL
LIN {X 0,Y 454.609,Z 625.954,A -85,B 0,C 180,E1 -8191.772,E2 -8191.772} C_VEL
LIN {X 0,Y 455.163,Z 618.732,A -85,B 0,C 180,E1 -8193.32,E2 -8193.32} C_VEL
LIN {X 0,Y 455.877,Z 610.034,A -85,B 0,C 180,E1 -8194.864,E2 -8194.864} C_VEL
LIN {X 0,Y 456.75,Z 599.555,A -85,B 0,C 180,E1 -8196.405,E2 -8196.405} C_VEL
LIN {X 0,Y 457.564,Z 587.816,A -85,B 0,C 180,E1 -8197.835,E2 -8197.835} C_VEL
LIN {X 0,Y 458.427,Z 575.847,A -85,B 0,C 180,E1 -8199.041,E2 -8199.041} C_VEL
LIN {X 0,Y 459.313,Z 562.637,A -85,B 0,C 180,E1 -8200.135,E2 -8200.135} C_VEL
LIN {X 0,Y 460.008,Z 549.711,A -85,B 0,C 180,E1 -8201.01,E2 -8201.01} C_VEL
LIN {X 0,Y 460.671,Z 535.242,A -85,B 0,C 180,E1 -8201.783,E2 -8201.783} C_VEL
LIN {X 0,Y 461.134,Z 519.549,A -85,B 0,C 180,E1 -8202.411,E2 -8202.411} C_VEL
LIN {X 0,Y 461.355,Z 504.532,A -85,B 0,C 180,E1 -8202.829,E2 -8202.829} C_VEL
LIN {X 0,Y 462.18,Z 427.238,A -85,B 0,C 180,E1 -8204.081,E2 -8204.081} C_VEL
LIN {X 0,Y 462.518,Z 395.306,A -85,B 0,C 180,E1 -8204.592,E2 -8204.592} C_VEL
LIN {X 0,Y 453.561,Z 375.062,A -85,B 0,C 180,E1 -8205.408,E2 -8205.408} C_VEL
LIN {X 0,Y 453.498,Z 374.621,A -85,B 0,C 180,E1 -8205.426,E2 -8205.426} C_VEL
LIN {X 0,Y 453.487,Z 374.623,A -85,B 0,C 180,E1 -8209.027,E2 -8209.027} C_VEL
LIN {X 0,Y 453.471,Z 374.622,A -85,B 0,C 180,E1 -8211.836,E2 -8211.836} C_VEL
LIN {X 0,Y 453.45,Z 374.628,A -85,B 0,C 180,E1 -8214.738,E2 -8214.738} C_VEL
LIN {X 0,Y 453.456,Z 374.624,A -85,B 0,C 180,E1 -8217.941,E2 -8217.941} C_VEL
LIN {X 0,Y 453.446,Z 374.618,A -85,B 0,C 180,E1 -8220.761,E2 -8220.761} C_VEL
LIN {X 0,Y 453.453,Z 374.621,A -85,B 0,C 180,E1 -8223.914,E2 -8223.914} C_VEL
LIN {X 0,Y 453.432,Z 374.629,A -85,B 0,C 180,E1 -8227.191,E2 -8227.191} C_VEL
LIN {X 0,Y 453.465,Z 374.619,A -85,B 0,C 180,E1 -8230.611,E2 -8230.611} C_VEL
LIN {X 0,Y 453.436,Z 374.622,A -85,B 0,C 180,E1 -8234.224,E2 -8234.224} C_VEL
LIN {X 0,Y 453.411,Z 374.632,A -85,B 0,C 180,E1 -8236.999,E2 -8236.999} C_VEL
LIN {X 0,Y 453.466,Z 374.627,A -85,B 0,C 180,E1 -8239.412,E2 -8239.412} C_VEL
LIN {X 0,Y 453.432,Z 374.625,A -85,B 0,C 180,E1 -8242.808,E2 -8242.808} C_VEL
LIN {X 0,Y 453.449,Z 374.618,A -85,B 0,C 180,E1 -8246.085,E2 -8246.085} C_VEL
LIN {X 0,Y 453.44,Z 374.631,A -85,B 0,C 180,E1 -8249.237,E2 -8249.237} C_VEL
LIN {X 0,Y 453.462,Z 374.62,A -85,B 0,C 180,E1 -8252.292,E2 -8252.292} C_VEL
LIN {X 0,Y 453.454,Z 374.625,A -85,B 0,C 180,E1 -8255.262,E2 -8255.262} C_VEL
LIN {X 0,Y 453.473,Z 374.62,A -85,B 0,C 180,E1 -8258.415,E2 -8258.415} C_VEL
LIN {X 0,Y 453.515,Z 374.615,A -85,B 0,C 180,E1 -8261.008,E2 -8261.008} C_VEL
LIN {X 0,Y 453.53,Z 374.614,A -85,B 0,C 180,E1 -8263.893,E2 -8263.893} C_VEL
LIN {X 0,Y 453.556,Z 374.597,A -85,B 0,C 180,E1 -8267.471,E2 -8267.471} C_VEL
LIN {X 0,Y 453.547,Z 374.597,A -85,B 0,C 180,E1 -8271.085,E2 -8271.085} C_VEL
LIN {X 0,Y 453.625,Z 374.605,A -85,B 0,C 180,E1 -8273.774,E2 -8273.774} C_VEL
LIN {X 0,Y 453.674,Z 374.595,A -85,B 0,C 180,E1 -8277.336,E2 -8277.336} C_VEL
LIN {X 0,Y 453.715,Z 374.591,A -85,B 0,C 180,E1 -8280,E2 -8280} C_VEL
LIN {X 0,Y 453.7,Z 374.588,A -85,B 0,C 180,E1 -8282.663,E2 -8282.663} C_VEL
LIN {X 0,Y 453.616,Z 374.602,A -85,B 0,C 180,E1 -8286.226,E2 -8286.226} C_VEL
LIN {X 0,Y 453.55,Z 374.606,A -85,B 0,C 180,E1 -8288.914,E2 -8288.914} C_VEL
LIN {X 0,Y 453.555,Z 374.609,A -85,B 0,C 180,E1 -8292.529,E2 -8292.529} C_VEL
LIN {X 0,Y 453.487,Z 374.62,A -85,B 0,C 180,E1 -8296.198,E2 -8296.198} C_VEL
LIN {X 0,Y 453.476,Z 374.616,A -85,B 0,C 180,E1 -8299.028,E2 -8299.028} C_VEL
LIN {X 0,Y 453.46,Z 374.625,A -85,B 0,C 180,E1 -8301.837,E2 -8301.837} C_VEL
LIN {X 0,Y 453.459,Z 374.622,A -85,B 0,C 180,E1 -8304.737,E2 -8304.737} C_VEL
LIN {X 0,Y 453.453,Z 374.628,A -85,B 0,C 180,E1 -8307.943,E2 -8307.943} C_VEL
LIN {X 0,Y 453.448,Z 374.624,A -85,B 0,C 180,E1 -8310.761,E2 -8310.761} C_VEL
LIN {X 0,Y 453.457,Z 374.619,A -85,B 0,C 180,E1 -8313.914,E2 -8313.914} C_VEL
LIN {X 0,Y 453.427,Z 374.629,A -85,B 0,C 180,E1 -8317.192,E2 -8317.192} C_VEL
LIN {X 0,Y 453.463,Z 374.622,A -85,B 0,C 180,E1 -8320.612,E2 -8320.612} C_VEL
LIN {X 0,Y 453.473,Z 374.621,A -85,B 0,C 180,E1 -8324.528,E2 -8324.528} C_VEL
LIN {X 0,Y 453.426,Z 374.623,A -85,B 0,C 180,E1 -8328.072,E2 -8328.072} C_VEL
LIN {X 0,Y 453.42,Z 374.628,A -85,B 0,C 180,E1 -8330.805,E2 -8330.805} C_VEL
LIN {X 0,Y 453.437,Z 374.628,A -85,B 0,C 180,E1 -8333.916,E2 -8333.916} C_VEL
LIN {X 0,Y 453.492,Z 374.78,A -85,B 0,C 180,E1 -8334.642,E2 -8334.642} C_VEL
LIN {X 0,Y 458.449,Z 393.398,A -85,B 0,C 180,E1 -8337.27,E2 -8337.27} C_VEL
LIN {X 0,Y 460.265,Z 401.344,A -85,B 0,C 180,E1 -8338.34,E2 -8338.34} C_VEL
LIN {X 0,Y 459.036,Z 424.137,A -85,B 0,C 180,E1 -8341.02,E2 -8341.02} C_VEL
LIN {X 0,Y 457.869,Z 448.164,A -85,B 0,C 180,E1 -8343.814,E2 -8343.814} C_VEL
LIN {X 0,Y 457.304,Z 459.841,A -85,B 0,C 180,E1 -8345.162,E2 -8345.162} C_VEL
LIN {X 0,Y 462.211,Z 494.419,A -85,B 0,C 180,E1 -8345.991,E2 -8345.991} C_VEL
LIN {X 0,Y 460.524,Z 629.097,A -85,B 0,C 180,E1 -8348.133,E2 -8348.133} C_VEL
LIN {X 0,Y 459.891,Z 645.072,A -85,B 0,C 180,E1 -8348.56,E2 -8348.56} C_VEL
LIN {X 0,Y 459.124,Z 659.012,A -85,B 0,C 180,E1 -8349.096,E2 -8349.096} C_VEL
LIN {X 0,Y 458.231,Z 673.234,A -85,B 0,C 180,E1 -8349.813,E2 -8349.813} C_VEL
LIN {X 0,Y 457.265,Z 687.207,A -85,B 0,C 180,E1 -8350.704,E2 -8350.704} C_VEL
LIN {X 0,Y 456.381,Z 700.083,A -85,B 0,C 180,E1 -8351.714,E2 -8351.714} C_VEL
LIN {X 0,Y 455.543,Z 712.067,A -85,B 0,C 180,E1 -8352.839,E2 -8352.839} C_VEL
LIN {X 0,Y 454.711,Z 723.213,A -85,B 0,C 180,E1 -8354.077,E2 -8354.077} C_VEL
LIN {X 0,Y 454.063,Z 733.553,A -85,B 0,C 180,E1 -8355.433,E2 -8355.433} C_VEL
LIN {X 0,Y 453.528,Z 743.69,A -85,B 0,C 180,E1 -8357.015,E2 -8357.015} C_VEL
LIN {X 0,Y 453.17,Z 752.163,A -85,B 0,C 180,E1 -8358.595,E2 -8358.595} C_VEL
LIN {X 0,Y 452.914,Z 759.165,A -85,B 0,C 180,E1 -8360.172,E2 -8360.172} C_VEL
LIN {X 0,Y 452.87,Z 765.675,A -85,B 0,C 180,E1 -8361.971,E2 -8361.971} C_VEL
LIN {X 0,Y 452.859,Z 770.71,A -85,B 0,C 180,E1 -8363.763,E2 -8363.763} C_VEL
LIN {X 0,Y 452.93,Z 774.407,A -85,B 0,C 180,E1 -8365.55,E2 -8365.55} C_VEL
LIN {X 0,Y 452.881,Z 776.818,A -85,B 0,C 180,E1 -8367.331,E2 -8367.331} C_VEL
LIN {X 0,Y 452.995,Z 778.042,A -85,B 0,C 180,E1 -8369.111,E2 -8369.111} C_VEL
LIN {X 0,Y 452.995,Z 778.019,A -85,B 0,C 180,E1 -8370.889,E2 -8370.889} C_VEL
LIN {X 0,Y 452.888,Z 776.758,A -85,B 0,C 180,E1 -8372.668,E2 -8372.668} C_VEL
LIN {X 0,Y 452.952,Z 774.316,A -85,B 0,C 180,E1 -8374.449,E2 -8374.449} C_VEL
LIN {X 0,Y 452.875,Z 770.597,A -85,B 0,C 180,E1 -8376.236,E2 -8376.236} C_VEL
LIN {X 0,Y 452.874,Z 765.545,A -85,B 0,C 180,E1 -8378.028,E2 -8378.028} C_VEL
LIN {X 0,Y 452.926,Z 759.028,A -85,B 0,C 180,E1 -8379.827,E2 -8379.827} C_VEL
LIN {X 0,Y 453.159,Z 752.019,A -85,B 0,C 180,E1 -8381.404,E2 -8381.404} C_VEL
LIN {X 0,Y 453.596,Z 742.294,A -85,B 0,C 180,E1 -8383.21,E2 -8383.21} C_VEL
LIN {X 0,Y 454.15,Z 731.98,A -85,B 0,C 180,E1 -8384.793,E2 -8384.793} C_VEL
LIN {X 0,Y 454.997,Z 720.053,A -85,B 0,C 180,E1 -8386.315,E2 -8386.315} C_VEL
LIN {X 0,Y 455.857,Z 707.93,A -85,B 0,C 180,E1 -8387.611,E2 -8387.611} C_VEL
LIN {X 0,Y 456.761,Z 695.357,A -85,B 0,C 180,E1 -8388.734,E2 -8388.734} C_VEL
LIN {X 0,Y 457.75,Z 681.69,A -85,B 0,C 180,E1 -8389.74,E2 -8389.74} C_VEL
LIN {X 0,Y 458.83,Z 666.607,A -85,B 0,C 180,E1 -8390.627,E2 -8390.627} C_VEL
LIN {X 0,Y 459.787,Z 651.176,A -85,B 0,C 180,E1 -8391.32,E2 -8391.32} C_VEL
LIN {X 0,Y 460.567,Z 636.242,A -85,B 0,C 180,E1 -8391.805,E2 -8391.805} C_VEL
LIN {X 0,Y 461.038,Z 620.696,A -85,B 0,C 180,E1 -8392.135,E2 -8392.135} C_VEL
LIN {X 0,Y 462.631,Z 493.767,A -85,B 0,C 180,E1 -8394.168,E2 -8394.168} C_VEL
LIN {X 0,Y 457.581,Z 458.999,A -85,B 0,C 180,E1 -8395.061,E2 -8395.061} C_VEL
LIN {X 0,Y 459.147,Z 430.412,A -85,B 0,C 180,E1 -8398.451,E2 -8398.451} C_VEL
LIN {X 0,Y 460.667,Z 405.198,A -85,B 0,C 180,E1 -8401.5,E2 -8401.5} C_VEL
LIN {X 0,Y 460.749,Z 401.141,A -85,B 0,C 180,E1 -8402.008,E2 -8402.008} C_VEL
LIN {X 0,Y 457.376,Z 388.029,A -85,B 0,C 180,E1 -8403.926,E2 -8403.926} C_VEL
LIN {X 0,Y 453.429,Z 374.622,A -85,B 0,C 180,E1 -8406.041,E2 -8406.041} C_VEL
LIN {X 0,Y 453.433,Z 374.629,A -85,B 0,C 180,E1 -8409.454,E2 -8409.454} C_VEL
LIN {X 0,Y 453.431,Z 374.63,A -85,B 0,C 180,E1 -8411.929,E2 -8411.929} C_VEL
LIN {X 0,Y 453.471,Z 374.61,A -85,B 0,C 180,E1 -8415.471,E2 -8415.471} C_VEL
LIN {X 0,Y 453.459,Z 374.621,A -85,B 0,C 180,E1 -8419.387,E2 -8419.387} C_VEL
LIN {X 0,Y 453.423,Z 374.628,A -85,B 0,C 180,E1 -8422.808,E2 -8422.808} C_VEL
LIN {X 0,Y 453.452,Z 374.627,A -85,B 0,C 180,E1 -8426.085,E2 -8426.085} C_VEL
LIN {X 0,Y 453.443,Z 374.622,A -85,B 0,C 180,E1 -8429.238,E2 -8429.238} C_VEL
LIN {X 0,Y 453.459,Z 374.626,A -85,B 0,C 180,E1 -8432.293,E2 -8432.293} C_VEL
LIN {X 0,Y 453.454,Z 374.622,A -85,B 0,C 180,E1 -8435.262,E2 -8435.262} C_VEL
LIN {X 0,Y 453.462,Z 374.626,A -85,B 0,C 180,E1 -8438.417,E2 -8438.417} C_VEL
LIN {X 0,Y 453.471,Z 374.623,A -85,B 0,C 180,E1 -8441.007,E2 -8441.007} C_VEL
LIN {X 0,Y 453.501,Z 374.62,A -85,B 0,C 180,E1 -8444.725,E2 -8444.725} C_VEL
LIN {X 0,Y 453.541,Z 374.619,A -85,B 0,C 180,E1 -8448.379,E2 -8448.379} C_VEL
LIN {X 0,Y 453.545,Z 374.613,A -85,B 0,C 180,E1 -8451.086,E2 -8451.086} C_VEL
LIN {X 0,Y 453.612,Z 374.599,A -85,B 0,C 180,E1 -8453.774,E2 -8453.774} C_VEL
LIN {X 0,Y 453.697,Z 374.587,A -85,B 0,C 180,E1 -8457.337,E2 -8457.337} C_VEL
LIN {X 0,Y 453.73,Z 374.589,A -85,B 0,C 180,E1 -8460,E2 -8460} C_VEL
LIN {X 0,Y 453.694,Z 374.598,A -85,B 0,C 180,E1 -8462.664,E2 -8462.664} C_VEL
LIN {X 0,Y 453.64,Z 374.589,A -85,B 0,C 180,E1 -8466.226,E2 -8466.226} C_VEL
LIN {X 0,Y 453.56,Z 374.608,A -85,B 0,C 180,E1 -8468.914,E2 -8468.914} C_VEL
LIN {X 0,Y 453.551,Z 374.61,A -85,B 0,C 180,E1 -8472.529,E2 -8472.529} C_VEL
LIN {X 0,Y 453.532,Z 374.608,A -85,B 0,C 180,E1 -8476.197,E2 -8476.197} C_VEL
LIN {X 0,Y 453.504,Z 374.613,A -85,B 0,C 180,E1 -8479.04,E2 -8479.04} C_VEL
LIN {X 0,Y 453.463,Z 374.613,A -85,B 0,C 180,E1 -8481.837,E2 -8481.837} C_VEL
LIN {X 0,Y 453.473,Z 374.625,A -85,B 0,C 180,E1 -8484.737,E2 -8484.737} C_VEL
LIN {X 0,Y 453.452,Z 374.619,A -85,B 0,C 180,E1 -8487.944,E2 -8487.944} C_VEL
LIN {X 0,Y 453.456,Z 374.625,A -85,B 0,C 180,E1 -8490.761,E2 -8490.761} C_VEL
LIN {X 0,Y 453.457,Z 374.624,A -85,B 0,C 180,E1 -8493.915,E2 -8493.915} C_VEL
LIN {X 0,Y 453.443,Z 374.624,A -85,B 0,C 180,E1 -8497.191,E2 -8497.191} C_VEL
LIN {X 0,Y 453.462,Z 374.62,A -85,B 0,C 180,E1 -8500.613,E2 -8500.613} C_VEL
LIN {X 0,Y 453.452,Z 374.617,A -85,B 0,C 180,E1 -8504.223,E2 -8504.223} C_VEL
LIN {X 0,Y 453.431,Z 374.626,A -85,B 0,C 180,E1 -8507.003,E2 -8507.003} C_VEL
LIN {X 0,Y 453.465,Z 374.621,A -85,B 0,C 180,E1 -8509.414,E2 -8509.414} C_VEL
LIN {X 0,Y 453.445,Z 374.626,A -85,B 0,C 180,E1 -8512.811,E2 -8512.811} C_VEL
LIN {X 0,Y 453.482,Z 374.623,A -85,B 0,C 180,E1 -8516.239,E2 -8516.239} C_VEL
LIN {X 0,Y 454.498,Z 377.472,A -85,B 0,C 180,E1 -8516.366,E2 -8516.366} C_VEL
LIN {X 0,Y 463.466,Z 395.727,A -85,B 0,C 180,E1 -8517.261,E2 -8517.261} C_VEL
LIN {X 0,Y 462.1,Z 502.811,A -85,B 0,C 180,E1 -8519.006,E2 -8519.006} C_VEL
LIN {X 0,Y 461.868,Z 518.43,A -85,B 0,C 180,E1 -8519.417,E2 -8519.417} C_VEL
LIN {X 0,Y 461.385,Z 533.53,A -85,B 0,C 180,E1 -8520.002,E2 -8520.002} C_VEL
LIN {X 0,Y 460.725,Z 548.483,A -85,B 0,C 180,E1 -8520.783,E2 -8520.783} C_VEL
LIN {X 0,Y 459.875,Z 562.568,A -85,B 0,C 180,E1 -8521.723,E2 -8521.723} C_VEL
LIN {X 0,Y 459.863,Z 562.966,A -85,B 0,C 180,E1 -8521.753,E2 -8521.753} C_VEL
LIN {X 0,Y 459.014,Z 568.046,A -85,B 0,C 180,E1 -8522.114,E2 -8522.114} C_VEL
LIN {X 0,Y 455.754,Z 576.298,A -85,B 0,C 180,E1 -8522.672,E2 -8522.672} C_VEL
LIN {X 0,Y 452.435,Z 584.277,A -85,B 0,C 180,E1 -8523.29,E2 -8523.29} C_VEL
LIN {X 0,Y 451.464,Z 588.807,A -85,B 0,C 180,E1 -8523.749,E2 -8523.749} C_VEL
LIN {X 0,Y 450.51,Z 599.701,A -85,B 0,C 180,E1 -8525.091,E2 -8525.091} C_VEL
LIN {X 0,Y 449.564,Z 609.385,A -85,B 0,C 180,E1 -8526.508,E2 -8526.508} C_VEL
LIN {X 0,Y 448.706,Z 618.769,A -85,B 0,C 180,E1 -8528.162,E2 -8528.162} C_VEL
LIN {X 0,Y 447.931,Z 626.485,A -85,B 0,C 180,E1 -8529.808,E2 -8529.808} C_VEL
LIN {X 0,Y 447.36,Z 633.594,A -85,B 0,C 180,E1 -8531.688,E2 -8531.688} C_VEL
LIN {X 0,Y 446.87,Z 639.274,A -85,B 0,C 180,E1 -8533.61,E2 -8533.61} C_VEL
LIN {X 0,Y 446.526,Z 643.279,A -85,B 0,C 180,E1 -8535.415,E2 -8535.415} C_VEL
LIN {X 0,Y 446.276,Z 646.462,A -85,B 0,C 180,E1 -8537.525,E2 -8537.525} C_VEL
LIN {X 0,Y 446.156,Z 647.869,A -85,B 0,C 180,E1 -8539.105,E2 -8539.105} C_VEL
LIN {X 0,Y 446.163,Z 648.427,A -85,B 0,C 180,E1 -8540.938,E2 -8540.938} C_VEL
LIN {X 0,Y 446.231,Z 647.788,A -85,B 0,C 180,E1 -8542.856,E2 -8542.856} C_VEL
LIN {X 0,Y 446.312,Z 646.161,A -85,B 0,C 180,E1 -8544.579,E2 -8544.579} C_VEL
LIN {X 0,Y 446.415,Z 643.372,A -85,B 0,C 180,E1 -8546.39,E2 -8546.39} C_VEL
LIN {X 0,Y 446.694,Z 639.389,A -85,B 0,C 180,E1 -8548.197,E2 -8548.197} C_VEL
LIN {X 0,Y 447.057,Z 634.141,A -85,B 0,C 180,E1 -8550,E2 -8550} C_VEL
LIN {X 0,Y 447.645,Z 627.459,A -85,B 0,C 180,E1 -8551.8,E2 -8551.8} C_VEL
LIN {X 0,Y 448.336,Z 619.156,A -85,B 0,C 180,E1 -8553.595,E2 -8553.595} C_VEL
LIN {X 0,Y 449.071,Z 610.352,A -85,B 0,C 180,E1 -8555.163,E2 -8555.163} C_VEL
LIN {X 0,Y 449.864,Z 601.374,A -85,B 0,C 180,E1 -8556.504,E2 -8556.504} C_VEL
LIN {X 0,Y 450.647,Z 590.77,A -85,B 0,C 180,E1 -8557.843,E2 -8557.843} C_VEL
LIN {X 0,Y 451.467,Z 579.185,A -85,B 0,C 180,E1 -8559.069,E2 -8559.069} C_VEL
LIN {X 0,Y 452.429,Z 566.465,A -85,B 0,C 180,E1 -8560.178,E2 -8560.178} C_VEL
LIN {X 0,Y 453.146,Z 554.133,A -85,B 0,C 180,E1 -8561.065,E2 -8561.065} C_VEL
LIN {X 0,Y 453.892,Z 539.701,A -85,B 0,C 180,E1 -8561.896,E2 -8561.896} C_VEL
LIN {X 0,Y 454.401,Z 524.546,A -85,B 0,C 180,E1 -8562.562,E2 -8562.562} C_VEL
LIN {X 0,Y 454.683,Z 509.375,A -85,B 0,C 180,E1 -8563.037,E2 -8563.037} C_VEL
LIN {X 0,Y 454.803,Z 490.439,A -85,B 0,C 180,E1 -8563.403,E2 -8563.403} C_VEL
LIN {X 0,Y 455.964,Z 397.268,A -85,B 0,C 180,E1 -8564.903,E2 -8564.903} C_VEL
LIN {X 0,Y 446.619,Z 376.337,A -85,B 0,C 180,E1 -8565.769,E2 -8565.769} C_VEL
LIN {X 0,Y 446.455,Z 375.497,A -85,B 0,C 180,E1 -8565.83,E2 -8565.83} C_VEL
LIN {X 0,Y 446.434,Z 375.502,A -85,B 0,C 180,E1 -8569.305,E2 -8569.305} C_VEL
LIN {X 0,Y 446.407,Z 375.502,A -85,B 0,C 180,E1 -8572.2,E2 -8572.2} C_VEL
LIN {X 0,Y 446.406,Z 375.507,A -85,B 0,C 180,E1 -8575.155,E2 -8575.155} C_VEL
LIN {X 0,Y 446.415,Z 375.501,A -85,B 0,C 180,E1 -8578.183,E2 -8578.183} C_VEL
LIN {X 0,Y 446.388,Z 375.506,A -85,B 0,C 180,E1 -8581.302,E2 -8581.302} C_VEL
LIN {X 0,Y 446.412,Z 375.499,A -85,B 0,C 180,E1 -8584.524,E2 -8584.524} C_VEL
LIN {X 0,Y 446.386,Z 375.504,A -85,B 0,C 180,E1 -8587.88,E2 -8587.88} C_VEL
LIN {X 0,Y 446.395,Z 375.502,A -85,B 0,C 180,E1 -8590.912,E2 -8590.912} C_VEL
LIN {X 0,Y 446.372,Z 375.503,A -85,B 0,C 180,E1 -8593.849,E2 -8593.849} C_VEL
LIN {X 0,Y 446.375,Z 375.504,A -85,B 0,C 180,E1 -8596.406,E2 -8596.406} C_VEL
LIN {X 0,Y 446.392,Z 375.504,A -85,B 0,C 180,E1 -8599.796,E2 -8599.796} C_VEL
LIN {X 0,Y 446.389,Z 375.508,A -85,B 0,C 180,E1 -8603.253,E2 -8603.253} C_VEL
LIN {X 0,Y 446.419,Z 375.494,A -85,B 0,C 180,E1 -8606.55,E2 -8606.55} C_VEL
LIN {X 0,Y 446.407,Z 375.498,A -85,B 0,C 180,E1 -8609.983,E2 -8609.983} C_VEL
LIN {X 0,Y 446.375,Z 375.505,A -85,B 0,C 180,E1 -8612.832,E2 -8612.832} C_VEL
LIN {X 0,Y 446.415,Z 375.496,A -85,B 0,C 180,E1 -8615.936,E2 -8615.936} C_VEL
LIN {X 0,Y 446.445,Z 375.497,A -85,B 0,C 180,E1 -8618.772,E2 -8618.772} C_VEL
LIN {X 0,Y 446.44,Z 375.498,A -85,B 0,C 180,E1 -8621.648,E2 -8621.648} C_VEL
LIN {X 0,Y 446.468,Z 375.492,A -85,B 0,C 180,E1 -8624.478,E2 -8624.478} C_VEL
LIN {X 0,Y 446.506,Z 375.467,A -85,B 0,C 180,E1 -8628.192,E2 -8628.192} C_VEL
LIN {X 0,Y 446.499,Z 375.473,A -85,B 0,C 180,E1 -8630.944,E2 -8630.944} C_VEL
LIN {X 0,Y 446.595,Z 375.482,A -85,B 0,C 180,E1 -8633.675,E2 -8633.675} C_VEL
LIN {X 0,Y 446.626,Z 375.472,A -85,B 0,C 180,E1 -8637.294,E2 -8637.294} C_VEL
LIN {X 0,Y 446.667,Z 375.469,A -85,B 0,C 180,E1 -8640,E2 -8640} C_VEL
LIN {X 0,Y 446.65,Z 375.466,A -85,B 0,C 180,E1 -8642.705,E2 -8642.705} C_VEL
LIN {X 0,Y 446.589,Z 375.477,A -85,B 0,C 180,E1 -8646.324,E2 -8646.324} C_VEL
LIN {X 0,Y 446.491,Z 375.491,A -85,B 0,C 180,E1 -8649.971,E2 -8649.971} C_VEL
LIN {X 0,Y 446.512,Z 375.486,A -85,B 0,C 180,E1 -8652.73,E2 -8652.73} C_VEL
LIN {X 0,Y 446.441,Z 375.498,A -85,B 0,C 180,E1 -8656.207,E2 -8656.207} C_VEL
LIN {X 0,Y 446.422,Z 375.497,A -85,B 0,C 180,E1 -8659.305,E2 -8659.305} C_VEL
LIN {X 0,Y 446.398,Z 375.5,A -85,B 0,C 180,E1 -8662.2,E2 -8662.2} C_VEL
LIN {X 0,Y 446.412,Z 375.501,A -85,B 0,C 180,E1 -8665.155,E2 -8665.155} C_VEL
LIN {X 0,Y 446.408,Z 375.502,A -85,B 0,C 180,E1 -8668.184,E2 -8668.184} C_VEL
LIN {X 0,Y 446.401,Z 375.504,A -85,B 0,C 180,E1 -8671.301,E2 -8671.301} C_VEL
LIN {X 0,Y 446.412,Z 375.498,A -85,B 0,C 180,E1 -8674.524,E2 -8674.524} C_VEL
LIN {X 0,Y 446.389,Z 375.5,A -85,B 0,C 180,E1 -8678.076,E2 -8678.076} C_VEL
LIN {X 0,Y 446.393,Z 375.506,A -85,B 0,C 180,E1 -8681.395,E2 -8681.395} C_VEL
LIN {X 0,Y 446.414,Z 375.5,A -85,B 0,C 180,E1 -8685.108,E2 -8685.108} C_VEL
LIN {X 0,Y 446.39,Z 375.494,A -85,B 0,C 180,E1 -8688.606,E2 -8688.606} C_VEL
LIN {X 0,Y 446.384,Z 375.509,A -85,B 0,C 180,E1 -8692.12,E2 -8692.12} C_VEL
LIN {X 0,Y 446.449,Z 375.684,A -85,B 0,C 180,E1 -8694.308,E2 -8694.308} C_VEL
LIN {X 0,Y 451.442,Z 394.286,A -85,B 0,C 180,E1 -8696.984,E2 -8696.984} C_VEL
LIN {X 0,Y 453.421,Z 402.154,A -85,B 0,C 180,E1 -8698.073,E2 -8698.073} C_VEL
LIN {X 0,Y 452.373,Z 422.075,A -85,B 0,C 180,E1 -8700.459,E2 -8700.459} C_VEL
LIN {X 0,Y 451.138,Z 445.825,A -85,B 0,C 180,E1 -8703.268,E2 -8703.268} C_VEL
LIN {X 0,Y 450.463,Z 458.974,A -85,B 0,C 180,E1 -8704.809,E2 -8704.809} C_VEL
LIN {X 0,Y 455.577,Z 496.053,A -85,B 0,C 180,E1 -8705.692,E2 -8705.692} C_VEL
LIN {X 0,Y 453.845,Z 628.263,A -85,B 0,C 180,E1 -8707.824,E2 -8707.824} C_VEL
LIN {X 0,Y 453.154,Z 644.379,A -85,B 0,C 180,E1 -8708.263,E2 -8708.263} C_VEL
LIN {X 0,Y 452.306,Z 659.373,A -85,B 0,C 180,E1 -8708.855,E2 -8708.855} C_VEL
LIN {X 0,Y 451.338,Z 673.81,A -85,B 0,C 180,E1 -8709.61,E2 -8709.61} C_VEL
LIN {X 0,Y 450.344,Z 687.482,A -85,B 0,C 180,E1 -8710.514,E2 -8710.514} C_VEL
LIN {X 0,Y 449.338,Z 701.451,A -85,B 0,C 180,E1 -8711.653,E2 -8711.653} C_VEL
LIN {X 0,Y 448.345,Z 714.77,A -85,B 0,C 180,E1 -8712.979,E2 -8712.979} C_VEL
LIN {X 0,Y 447.548,Z 725.719,A -85,B 0,C 180,E1 -8714.283,E2 -8714.283} C_VEL
LIN {X 0,Y 446.809,Z 737.01,A -85,B 0,C 180,E1 -8715.889,E2 -8715.889} C_VEL
LIN {X 0,Y 446.286,Z 746.524,A -85,B 0,C 180,E1 -8717.516,E2 -8717.516} C_VEL
LIN {X 0,Y 446.045,Z 754.233,A -85,B 0,C 180,E1 -8719.101,E2 -8719.101} C_VEL
LIN {X 0,Y 445.811,Z 761.544,A -85,B 0,C 180,E1 -8720.93,E2 -8720.93} C_VEL
LIN {X 0,Y 445.797,Z 767.317,A -85,B 0,C 180,E1 -8722.754,E2 -8722.754} C_VEL
LIN {X 0,Y 445.821,Z 771.682,A -85,B 0,C 180,E1 -8724.572,E2 -8724.572} C_VEL
LIN {X 0,Y 445.837,Z 774.737,A -85,B 0,C 180,E1 -8726.385,E2 -8726.385} C_VEL
LIN {X 0,Y 445.834,Z 776.551,A -85,B 0,C 180,E1 -8728.193,E2 -8728.193} C_VEL
LIN {X 0,Y 445.977,Z 777.028,A -85,B 0,C 180,E1 -8729.097,E2 -8729.097} C_VEL
LIN {X 0,Y 445.978,Z 777.006,A -85,B 0,C 180,E1 -8730.903,E2 -8730.903} C_VEL
LIN {X 0,Y 445.849,Z 775.745,A -85,B 0,C 180,E1 -8732.71,E2 -8732.71} C_VEL
LIN {X 0,Y 445.894,Z 773.304,A -85,B 0,C 180,E1 -8734.52,E2 -8734.52} C_VEL
LIN {X 0,Y 445.834,Z 769.592,A -85,B 0,C 180,E1 -8736.335,E2 -8736.335} C_VEL
LIN {X 0,Y 445.808,Z 764.544,A -85,B 0,C 180,E1 -8738.156,E2 -8738.156} C_VEL
LIN {X 0,Y 445.875,Z 758.038,A -85,B 0,C 180,E1 -8739.984,E2 -8739.984} C_VEL
LIN {X 0,Y 446.103,Z 751.036,A -85,B 0,C 180,E1 -8741.587,E2 -8741.587} C_VEL
LIN {X 0,Y 446.492,Z 742.627,A -85,B 0,C 180,E1 -8743.193,E2 -8743.193} C_VEL
LIN {X 0,Y 447.071,Z 732.599,A -85,B 0,C 180,E1 -8744.8,E2 -8744.8} C_VEL
LIN {X 0,Y 447.773,Z 722.418,A -85,B 0,C 180,E1 -8746.176,E2 -8746.176} C_VEL
LIN {X 0,Y 448.745,Z 710.402,A -85,B 0,C 180,E1 -8747.546,E2 -8747.546} C_VEL
LIN {X 0,Y 449.739,Z 697.195,A -85,B 0,C 180,E1 -8748.801,E2 -8748.801} C_VEL
LIN {X 0,Y 450.753,Z 684.172,A -85,B 0,C 180,E1 -8749.822,E2 -8749.822} C_VEL
LIN {X 0,Y 451.882,Z 670.02,A -85,B 0,C 180,E1 -8750.72,E2 -8750.72} C_VEL
LIN {X 0,Y 452.891,Z 655.035,A -85,B 0,C 180,E1 -8751.467,E2 -8751.467} C_VEL
LIN {X 0,Y 453.783,Z 639.727,A -85,B 0,C 180,E1 -8752.029,E2 -8752.029} C_VEL
LIN {X 0,Y 454.4,Z 624.07,A -85,B 0,C 180,E1 -8752.416,E2 -8752.416} C_VEL
LIN {X 0,Y 456.204,Z 494.77,A -85,B 0,C 180,E1 -8754.526,E2 -8754.526} C_VEL
LIN {X 0,Y 451.296,Z 460.793,A -85,B 0,C 180,E1 -8755.414,E2 -8755.414} C_VEL
LIN {X 0,Y 450.831,Z 457.858,A -85,B 0,C 180,E1 -8755.502,E2 -8755.502} C_VEL
LIN {X 0,Y 452.426,Z 430.668,A -85,B 0,C 180,E1 -8758.786,E2 -8758.786} C_VEL
LIN {X 0,Y 454.007,Z 406.516,A -85,B 0,C 180,E1 -8761.756,E2 -8761.756} C_VEL
LIN {X 0,Y 453.939,Z 402.457,A -85,B 0,C 180,E1 -8762.284,E2 -8762.284} C_VEL
LIN {X 0,Y 449.823,Z 386.804,A -85,B 0,C 180,E1 -8764.64,E2 -8764.64} C_VEL
LIN {X 0,Y 446.393,Z 375.498,A -85,B 0,C 180,E1 -8766.466,E2 -8766.466} C_VEL
LIN {X 0,Y 446.386,Z 375.506,A -85,B 0,C 180,E1 -8769.515,E2 -8769.515} C_VEL
LIN {X 0,Y 446.37,Z 375.506,A -85,B 0,C 180,E1 -8772.61,E2 -8772.61} C_VEL
LIN {X 0,Y 446.411,Z 375.49,A -85,B 0,C 180,E1 -8775.107,E2 -8775.107} C_VEL
LIN {X 0,Y 446.389,Z 375.503,A -85,B 0,C 180,E1 -8778.605,E2 -8778.605} C_VEL
LIN {X 0,Y 446.386,Z 375.504,A -85,B 0,C 180,E1 -8781.923,E2 -8781.923} C_VEL
LIN {X 0,Y 446.407,Z 375.502,A -85,B 0,C 180,E1 -8785.475,E2 -8785.475} C_VEL
LIN {X 0,Y 446.396,Z 375.503,A -85,B 0,C 180,E1 -8788.698,E2 -8788.698} C_VEL
LIN {X 0,Y 446.411,Z 375.504,A -85,B 0,C 180,E1 -8791.836,E2 -8791.836} C_VEL
LIN {X 0,Y 446.407,Z 375.502,A -85,B 0,C 180,E1 -8794.845,E2 -8794.845} C_VEL
LIN {X 0,Y 446.43,Z 375.504,A -85,B 0,C 180,E1 -8798.246,E2 -8798.246} C_VEL
LIN {X 0,Y 446.397,Z 375.503,A -85,B 0,C 180,E1 -8801.647,E2 -8801.647} C_VEL
LIN {X 0,Y 446.442,Z 375.503,A -85,B 0,C 180,E1 -8804.478,E2 -8804.478} C_VEL
LIN {X 0,Y 446.502,Z 375.489,A -85,B 0,C 180,E1 -8807.384,E2 -8807.384} C_VEL
LIN {X 0,Y 446.496,Z 375.492,A -85,B 0,C 180,E1 -8810.944,E2 -8810.944} C_VEL
LIN {X 0,Y 446.583,Z 375.474,A -85,B 0,C 180,E1 -8813.676,E2 -8813.676} C_VEL
LIN {X 0,Y 446.647,Z 375.466,A -85,B 0,C 180,E1 -8817.295,E2 -8817.295} C_VEL
LIN {X 0,Y 446.682,Z 375.467,A -85,B 0,C 180,E1 -8820,E2 -8820} C_VEL
LIN {X 0,Y 446.643,Z 375.477,A -85,B 0,C 180,E1 -8822.706,E2 -8822.706} C_VEL
LIN {X 0,Y 446.609,Z 375.462,A -85,B 0,C 180,E1 -8826.324,E2 -8826.324} C_VEL
LIN {X 0,Y 446.508,Z 375.489,A -85,B 0,C 180,E1 -8829.056,E2 -8829.056} C_VEL
LIN {X 0,Y 446.509,Z 375.483,A -85,B 0,C 180,E1 -8832.73,E2 -8832.73} C_VEL
LIN {X 0,Y 446.476,Z 375.489,A -85,B 0,C 180,E1 -8836.46,E2 -8836.46} C_VEL
LIN {X 0,Y 446.456,Z 375.489,A -85,B 0,C 180,E1 -8839.304,E2 -8839.304} C_VEL
LIN {X 0,Y 446.404,Z 375.494,A -85,B 0,C 180,E1 -8842.201,E2 -8842.201} C_VEL
LIN {X 0,Y 446.417,Z 375.497,A -85,B 0,C 180,E1 -8845.155,E2 -8845.155} C_VEL
LIN {X 0,Y 446.426,Z 375.495,A -85,B 0,C 180,E1 -8848.183,E2 -8848.183} C_VEL
LIN {X 0,Y 446.401,Z 375.495,A -85,B 0,C 180,E1 -8851.302,E2 -8851.302} C_VEL
LIN {X 0,Y 446.413,Z 375.505,A -85,B 0,C 180,E1 -8854.525,E2 -8854.525} C_VEL
LIN {X 0,Y 446.403,Z 375.502,A -85,B 0,C 180,E1 -8858.08,E2 -8858.08} C_VEL
LIN {X 0,Y 446.394,Z 375.505,A -85,B 0,C 180,E1 -8861.395,E2 -8861.395} C_VEL
LIN {X 0,Y 446.443,Z 375.5,A -85,B 0,C 180,E1 -8865.105,E2 -8865.105} C_VEL
LIN {X 0,Y 446.401,Z 375.505,A -85,B 0,C 180,E1 -8868.608,E2 -8868.608} C_VEL
LIN {X 0,Y 446.405,Z 375.498,A -85,B 0,C 180,E1 -8871.923,E2 -8871.923} C_VEL
LIN {X 0,Y 446.42,Z 375.504,A -85,B 0,C 180,E1 -8875.478,E2 -8875.478} C_VEL
LIN {X 0,Y 446.435,Z 375.535,A -85,B 0,C 180,E1 -8875.785,E2 -8875.785} C_VEL
LIN {X 0,Y 447.5,Z 378.441,A -85,B 0,C 180,E1 -8875.91,E2 -8875.91} C_VEL
LIN {X 0,Y 455.892,Z 395.115,A -85,B 0,C 180,E1 -8876.766,E2 -8876.766} C_VEL
LIN {X 0,Y 457.143,Z 397.794,A -85,B 0,C 180,E1 -8876.894,E2 -8876.894} C_VEL
LIN {X 0,Y 455.674,Z 503.937,A -85,B 0,C 180,E1 -8878.649,E2 -8878.649} C_VEL
LIN {X 0,Y 455.431,Z 519.518,A -85,B 0,C 180,E1 -8879.066,E2 -8879.066} C_VEL
LIN {X 0,Y 454.987,Z 533.543,A -85,B 0,C 180,E1 -8879.613,E2 -8879.613} C_VEL
LIN {X 0,Y 454.284,Z 548.517,A -85,B 0,C 180,E1 -8880.392,E2 -8880.392} C_VEL
LIN {X 0,Y 453.468,Z 561.995,A -85,B 0,C 180,E1 -8881.287,E2 -8881.287} C_VEL
LIN {X 0,Y 452.604,Z 574.835,A -85,B 0,C 180,E1 -8882.341,E2 -8882.341} C_VEL
LIN {X 0,Y 451.623,Z 586.979,A -85,B 0,C 180,E1 -8883.549,E2 -8883.549} C_VEL
LIN {X 0,Y 451.464,Z 588.807,A -85,B 0,C 180,E1 -8883.749,E2 -8883.749} C_VEL
LIN {X 0,Y 450.532,Z 593.261,A -85,B 0,C 180,E1 -8884.227,E2 -8884.227} C_VEL
LIN {X 0,Y 447.218,Z 600.463,A -85,B 0,C 180,E1 -8884.987,E2 -8884.987} C_VEL
LIN {X 0,Y 443.81,Z 607.35,A -85,B 0,C 180,E1 -8885.805,E2 -8885.805} C_VEL
LIN {X 0,Y 442.746,Z 611.132,A -85,B 0,C 180,E1 -8886.368,E2 -8886.368} C_VEL
LIN {X 0,Y 441.84,Z 620.408,A -85,B 0,C 180,E1 -8888.051,E2 -8888.051} C_VEL
LIN {X 0,Y 440.976,Z 628.73,A -85,B 0,C 180,E1 -8889.896,E2 -8889.896} C_VEL
LIN {X 0,Y 440.481,Z 634.22,A -85,B 0,C 180,E1 -8891.392,E2 -8891.392} C_VEL
LIN {X 0,Y 439.935,Z 639.854,A -85,B 0,C 180,E1 -8893.289,E2 -8893.289} C_VEL
LIN {X 0,Y 439.555,Z 644.083,A -85,B 0,C 180,E1 -8895.178,E2 -8895.178} C_VEL
LIN {X 0,Y 439.303,Z 647.044,A -85,B 0,C 180,E1 -8897.058,E2 -8897.058} C_VEL
LIN {X 0,Y 439.148,Z 648.827,A -85,B 0,C 180,E1 -8898.929,E2 -8898.929} C_VEL
LIN {X 0,Y 439.149,Z 649.424,A -85,B 0,C 180,E1 -8900.792,E2 -8900.792} C_VEL
LIN {X 0,Y 439.196,Z 648.831,A -85,B 0,C 180,E1 -8902.806,E2 -8902.806} C_VEL
LIN {X 0,Y 439.303,Z 647.31,A -85,B 0,C 180,E1 -8904.492,E2 -8904.492} C_VEL
LIN {X 0,Y 439.381,Z 644.606,A -85,B 0,C 180,E1 -8906.332,E2 -8906.332} C_VEL
LIN {X 0,Y 439.689,Z 640.703,A -85,B 0,C 180,E1 -8908.168,E2 -8908.168} C_VEL
LIN {X 0,Y 440.057,Z 635.542,A -85,B 0,C 180,E1 -8910,E2 -8910} C_VEL
LIN {X 0,Y 440.688,Z 628.945,A -85,B 0,C 180,E1 -8911.828,E2 -8911.828} C_VEL
LIN {X 0,Y 441.387,Z 620.757,A -85,B 0,C 180,E1 -8913.652,E2 -8913.652} C_VEL
LIN {X 0,Y 442.167,Z 612.054,A -85,B 0,C 180,E1 -8915.244,E2 -8915.244} C_VEL
LIN {X 0,Y 443.11,Z 601.572,A -85,B 0,C 180,E1 -8916.832,E2 -8916.832} C_VEL
LIN {X 0,Y 444.042,Z 589.815,A -85,B 0,C 180,E1 -8918.304,E2 -8918.304} C_VEL
LIN {X 0,Y 444.826,Z 579.038,A -85,B 0,C 180,E1 -8919.435,E2 -8919.435} C_VEL
LIN {X 0,Y 445.809,Z 566.074,A -85,B 0,C 180,E1 -8920.56,E2 -8920.56} C_VEL
LIN {X 0,Y 446.571,Z 553.397,A -85,B 0,C 180,E1 -8921.46,E2 -8921.46} C_VEL
LIN {X 0,Y 447.342,Z 538.477,A -85,B 0,C 180,E1 -8922.303,E2 -8922.303} C_VEL
LIN {X 0,Y 447.82,Z 523.694,A -85,B 0,C 180,E1 -8922.936,E2 -8922.936} C_VEL
LIN {X 0,Y 448.095,Z 508.478,A -85,B 0,C 180,E1 -8923.395,E2 -8923.395} C_VEL
LIN {X 0,Y 448.298,Z 482.664,A -85,B 0,C 180,E1 -8923.861,E2 -8923.861} C_VEL
LIN {X 0,Y 449.373,Z 398.996,A -85,B 0,C 180,E1 -8925.228,E2 -8925.228} C_VEL
LIN {X 0,Y 439.502,Z 376.881,A -85,B 0,C 180,E1 -8926.165,E2 -8926.165} C_VEL
LIN {X 0,Y 439.422,Z 376.373,A -85,B 0,C 180,E1 -8926.195,E2 -8926.195} C_VEL
LIN {X 0,Y 439.38,Z 376.378,A -85,B 0,C 180,E1 -8929.627,E2 -8929.627} C_VEL
LIN {X 0,Y 439.351,Z 376.383,A -85,B 0,C 180,E1 -8932.576,E2 -8932.576} C_VEL
LIN {X 0,Y 439.35,Z 376.383,A -85,B 0,C 180,E1 -8935.588,E2 -8935.588} C_VEL
LIN {X 0,Y 439.376,Z 376.381,A -85,B 0,C 180,E1 -8938.676,E2 -8938.676} C_VEL
LIN {X 0,Y 439.341,Z 376.382,A -85,B 0,C 180,E1 -8942.024,E2 -8942.024} C_VEL
LIN {X 0,Y 439.383,Z 376.38,A -85,B 0,C 180,E1 -8945.338,E2 -8945.338} C_VEL
LIN {X 0,Y 439.348,Z 376.381,A -85,B 0,C 180,E1 -8948.598,E2 -8948.598} C_VEL
LIN {X 0,Y 439.358,Z 376.384,A -85,B 0,C 180,E1 -8951.252,E2 -8951.252} C_VEL
LIN {X 0,Y 439.364,Z 376.377,A -85,B 0,C 180,E1 -8954.733,E2 -8954.733} C_VEL
LIN {X 0,Y 439.343,Z 376.38,A -85,B 0,C 180,E1 -8957.789,E2 -8957.789} C_VEL
LIN {X 0,Y 439.349,Z 376.381,A -85,B 0,C 180,E1 -8961.401,E2 -8961.401} C_VEL
LIN {X 0,Y 439.385,Z 376.378,A -85,B 0,C 180,E1 -8964.842,E2 -8964.842} C_VEL
LIN {X 0,Y 439.339,Z 376.382,A -85,B 0,C 180,E1 -8968.136,E2 -8968.136} C_VEL
LIN {X 0,Y 439.37,Z 376.378,A -85,B 0,C 180,E1 -8971.323,E2 -8971.323} C_VEL
LIN {X 0,Y 439.346,Z 376.379,A -85,B 0,C 180,E1 -8974.411,E2 -8974.411} C_VEL
LIN {X 0,Y 439.354,Z 376.383,A -85,B 0,C 180,E1 -8977.424,E2 -8977.424} C_VEL
LIN {X 0,Y 439.434,Z 376.366,A -85,B 0,C 180,E1 -8980.663,E2 -8980.663} C_VEL
LIN {X 0,Y 439.436,Z 376.368,A -85,B 0,C 180,E1 -8984.223,E2 -8984.223} C_VEL
LIN {X 0,Y 439.473,Z 376.344,A -85,B 0,C 180,E1 -8988.001,E2 -8988.001} C_VEL
LIN {X 0,Y 439.47,Z 376.359,A -85,B 0,C 180,E1 -8991.725,E2 -8991.725} C_VEL
LIN {X 0,Y 439.585,Z 376.35,A -85,B 0,C 180,E1 -8994.495,E2 -8994.495} C_VEL
LIN {X 0,Y 439.611,Z 376.341,A -85,B 0,C 180,E1 -8998.167,E2 -8998.167} C_VEL
LIN {X 0,Y 439.619,Z 376.347,A -85,B 0,C 180,E1 -9000,E2 -9000} C_VEL
LIN {X 0,Y 439.602,Z 376.344,A -85,B 0,C 180,E1 -9002.749,E2 -9002.749} C_VEL
LIN {X 0,Y 439.543,Z 376.354,A -85,B 0,C 180,E1 -9006.426,E2 -9006.426} C_VEL
LIN {X 0,Y 439.467,Z 376.363,A -85,B 0,C 180,E1 -9009.202,E2 -9009.202} C_VEL
LIN {X 0,Y 439.455,Z 376.366,A -85,B 0,C 180,E1 -9012.938,E2 -9012.938} C_VEL
LIN {X 0,Y 439.387,Z 376.376,A -85,B 0,C 180,E1 -9016.325,E2 -9016.325} C_VEL
LIN {X 0,Y 439.368,Z 376.379,A -85,B 0,C 180,E1 -9019.628,E2 -9019.628} C_VEL
LIN {X 0,Y 439.343,Z 376.377,A -85,B 0,C 180,E1 -9022.576,E2 -9022.576} C_VEL
LIN {X 0,Y 439.358,Z 376.384,A -85,B 0,C 180,E1 -9025.588,E2 -9025.588} C_VEL
LIN {X 0,Y 439.373,Z 376.376,A -85,B 0,C 180,E1 -9028.676,E2 -9028.676} C_VEL
LIN {X 0,Y 439.357,Z 376.38,A -85,B 0,C 180,E1 -9032.029,E2 -9032.029} C_VEL
LIN {X 0,Y 439.379,Z 376.376,A -85,B 0,C 180,E1 -9035.339,E2 -9035.339} C_VEL
LIN {X 0,Y 439.346,Z 376.374,A -85,B 0,C 180,E1 -9038.599,E2 -9038.599} C_VEL
LIN {X 0,Y 439.356,Z 376.381,A -85,B 0,C 180,E1 -9041.253,E2 -9041.253} C_VEL
LIN {X 0,Y 439.368,Z 376.377,A -85,B 0,C 180,E1 -9044.733,E2 -9044.733} C_VEL
LIN {X 0,Y 439.34,Z 376.382,A -85,B 0,C 180,E1 -9047.79,E2 -9047.79} C_VEL
LIN {X 0,Y 439.344,Z 376.383,A -85,B 0,C 180,E1 -9051.402,E2 -9051.402} C_VEL
LIN {X 0,Y 439.385,Z 376.575,A -85,B 0,C 180,E1 -9053.958,E2 -9053.958} C_VEL
LIN {X 0,Y 444.036,Z 393.667,A -85,B 0,C 180,E1 -9056.476,E2 -9056.476} C_VEL
LIN {X 0,Y 446.673,Z 404.577,A -85,B 0,C 180,E1 -9058.009,E2 -9058.009} C_VEL
LIN {X 0,Y 445.257,Z 427.907,A -85,B 0,C 180,E1 -9060.835,E2 -9060.835} C_VEL
LIN {X 0,Y 444.066,Z 449.651,A -85,B 0,C 180,E1 -9063.443,E2 -9063.443} C_VEL
LIN {X 0,Y 443.599,Z 457.896,A -85,B 0,C 180,E1 -9064.425,E2 -9064.425} C_VEL
LIN {X 0,Y 448.971,Z 496.48,A -85,B 0,C 180,E1 -9065.367,E2 -9065.367} C_VEL
LIN {X 0,Y 447.183,Z 627.296,A -85,B 0,C 180,E1 -9067.506,E2 -9067.506} C_VEL
LIN {X 0,Y 446.485,Z 643.436,A -85,B 0,C 180,E1 -9067.953,E2 -9067.953} C_VEL
LIN {X 0,Y 445.604,Z 657.711,A -85,B 0,C 180,E1 -9068.519,E2 -9068.519} C_VEL
LIN {X 0,Y 444.604,Z 672.341,A -85,B 0,C 180,E1 -9069.287,E2 -9069.287} C_VEL
LIN {X 0,Y 443.515,Z 686.092,A -85,B 0,C 180,E1 -9070.202,E2 -9070.202} C_VEL
LIN {X 0,Y 442.532,Z 698.813,A -85,B 0,C 180,E1 -9071.241,E2 -9071.241} C_VEL
LIN {X 0,Y 441.548,Z 711.697,A -85,B 0,C 180,E1 -9072.507,E2 -9072.507} C_VEL
LIN {X 0,Y 440.669,Z 722.661,A -85,B 0,C 180,E1 -9073.794,E2 -9073.794} C_VEL
LIN {X 0,Y 439.945,Z 732.767,A -85,B 0,C 180,E1 -9075.191,E2 -9075.191} C_VEL
LIN {X 0,Y 439.393,Z 742.709,A -85,B 0,C 180,E1 -9076.825,E2 -9076.825} C_VEL
LIN {X 0,Y 439.007,Z 751.008,A -85,B 0,C 180,E1 -9078.457,E2 -9078.457} C_VEL
LIN {X 0,Y 438.816,Z 756.992,A -85,B 0,C 180,E1 -9079.853,E2 -9079.853} C_VEL
LIN {X 0,Y 438.723,Z 763.538,A -85,B 0,C 180,E1 -9081.71,E2 -9081.71} C_VEL
LIN {X 0,Y 438.759,Z 768.615,A -85,B 0,C 180,E1 -9083.562,E2 -9083.562} C_VEL
LIN {X 0,Y 438.817,Z 772.334,A -85,B 0,C 180,E1 -9085.407,E2 -9085.407} C_VEL
LIN {X 0,Y 438.806,Z 774.77,A -85,B 0,C 180,E1 -9087.246,E2 -9087.246} C_VEL
LIN {X 0,Y 438.958,Z 776.013,A -85,B 0,C 180,E1 -9089.082,E2 -9089.082} C_VEL
LIN {X 0,Y 438.959,Z 775.993,A -85,B 0,C 180,E1 -9090.917,E2 -9090.917} C_VEL
LIN {X 0,Y 438.81,Z 774.736,A -85,B 0,C 180,E1 -9092.754,E2 -9092.754} C_VEL
LIN {X 0,Y 438.837,Z 772.299,A -85,B 0,C 180,E1 -9094.592,E2 -9094.592} C_VEL
LIN {X 0,Y 438.794,Z 768.598,A -85,B 0,C 180,E1 -9096.437,E2 -9096.437} C_VEL
LIN {X 0,Y 438.727,Z 763.554,A -85,B 0,C 180,E1 -9098.289,E2 -9098.289} C_VEL
LIN {X 0,Y 438.816,Z 757.064,A -85,B 0,C 180,E1 -9100.146,E2 -9100.146} C_VEL
LIN {X 0,Y 439.04,Z 750.069,A -85,B 0,C 180,E1 -9101.776,E2 -9101.776} C_VEL
LIN {X 0,Y 439.554,Z 740.402,A -85,B 0,C 180,E1 -9103.64,E2 -9103.64} C_VEL
LIN {X 0,Y 440.204,Z 730.151,A -85,B 0,C 180,E1 -9105.273,E2 -9105.273} C_VEL
LIN {X 0,Y 441.163,Z 718.317,A -85,B 0,C 180,E1 -9106.842,E2 -9106.842} C_VEL
LIN {X 0,Y 442.134,Z 706.288,A -85,B 0,C 180,E1 -9108.176,E2 -9108.176} C_VEL
LIN {X 0,Y 443.273,Z 692.433,A -85,B 0,C 180,E1 -9109.447,E2 -9109.447} C_VEL
LIN {X 0,Y 444.449,Z 678.634,A -85,B 0,C 180,E1 -9110.478,E2 -9110.478} C_VEL
LIN {X 0,Y 445.613,Z 664.035,A -85,B 0,C 180,E1 -9111.349,E2 -9111.349} C_VEL
LIN {X 0,Y 446.644,Z 648.828,A -85,B 0,C 180,E1 -9112.047,E2 -9112.047} C_VEL
LIN {X 0,Y 447.575,Z 632.955,A -85,B 0,C 180,E1 -9112.564,E2 -9112.564} C_VEL
LIN {X 0,Y 448.059,Z 618.525,A -85,B 0,C 180,E1 -9112.873,E2 -9112.873} C_VEL
LIN {X 0,Y 449.783,Z 495.88,A -85,B 0,C 180,E1 -9114.896,E2 -9114.896} C_VEL
LIN {X 0,Y 445.095,Z 462.785,A -85,B 0,C 180,E1 -9115.777,E2 -9115.777} C_VEL
LIN {X 0,Y 444.072,Z 456.654,A -85,B 0,C 180,E1 -9115.97,E2 -9115.97} C_VEL
LIN {X 0,Y 445.808,Z 429.934,A -85,B 0,C 180,E1 -9119.254,E2 -9119.254} C_VEL
LIN {X 0,Y 447.414,Z 407.046,A -85,B 0,C 180,E1 -9122.12,E2 -9122.12} C_VEL
LIN {X 0,Y 447.109,Z 404.029,A -85,B 0,C 180,E1 -9122.538,E2 -9122.538} C_VEL
LIN {X 0,Y 443.246,Z 389.252,A -85,B 0,C 180,E1 -9124.805,E2 -9124.805} C_VEL
LIN {X 0,Y 439.327,Z 376.38,A -85,B 0,C 180,E1 -9126.93,E2 -9126.93} C_VEL
LIN {X 0,Y 439.337,Z 376.385,A -85,B 0,C 180,E1 -9129.839,E2 -9129.839} C_VEL
LIN {X 0,Y 439.327,Z 376.383,A -85,B 0,C 180,E1 -9132.619,E2 -9132.619} C_VEL
LIN {X 0,Y 439.365,Z 376.366,A -85,B 0,C 180,E1 -9135.266,E2 -9135.266} C_VEL
LIN {X 0,Y 439.342,Z 376.38,A -85,B 0,C 180,E1 -9139.015,E2 -9139.015} C_VEL
LIN {X 0,Y 439.344,Z 376.378,A -85,B 0,C 180,E1 -9141.61,E2 -9141.61} C_VEL
LIN {X 0,Y 439.379,Z 376.379,A -85,B 0,C 180,E1 -9144.842,E2 -9144.842} C_VEL
LIN {X 0,Y 439.356,Z 376.385,A -85,B 0,C 180,E1 -9148.138,E2 -9148.138} C_VEL
LIN {X 0,Y 439.374,Z 376.379,A -85,B 0,C 180,E1 -9151.609,E2 -9151.609} C_VEL
LIN {X 0,Y 439.353,Z 376.386,A -85,B 0,C 180,E1 -9154.412,E2 -9154.412} C_VEL
LIN {X 0,Y 439.339,Z 376.383,A -85,B 0,C 180,E1 -9157.423,E2 -9157.423} C_VEL
LIN {X 0,Y 439.371,Z 376.383,A -85,B 0,C 180,E1 -9160.684,E2 -9160.684} C_VEL
LIN {X 0,Y 439.401,Z 376.378,A -85,B 0,C 180,E1 -9164.222,E2 -9164.222} C_VEL
LIN {X 0,Y 439.471,Z 376.365,A -85,B 0,C 180,E1 -9167.285,E2 -9167.285} C_VEL
LIN {X 0,Y 439.463,Z 376.37,A -85,B 0,C 180,E1 -9170.798,E2 -9170.798} C_VEL
LIN {X 0,Y 439.535,Z 376.352,A -85,B 0,C 180,E1 -9173.574,E2 -9173.574} C_VEL
LIN {X 0,Y 439.394,Z 376.374,A -85,B 0,C 180,E1 -9175.413,E2 -9175.413} C_VEL
LIN {X 0,Y 439.615,Z 376.344,A -85,B 0,C 180,E1 -9178.168,E2 -9178.168} C_VEL
LIN {X 0,Y 439.581,Z 376.349,A -85,B 0,C 180,E1 -9180.916,E2 -9180.916} C_VEL
LIN {X 0,Y 439.595,Z 376.355,A -85,B 0,C 180,E1 -9182.749,E2 -9182.749} C_VEL
LIN {X 0,Y 439.581,Z 376.336,A -85,B 0,C 180,E1 -9186.426,E2 -9186.426} C_VEL
LIN {X 0,Y 439.472,Z 376.364,A -85,B 0,C 180,E1 -9189.202,E2 -9189.202} C_VEL
LIN {X 0,Y 439.452,Z 376.358,A -85,B 0,C 180,E1 -9192.938,E2 -9192.938} C_VEL
LIN {X 0,Y 439.434,Z 376.365,A -85,B 0,C 180,E1 -9196.349,E2 -9196.349} C_VEL
LIN {X 0,Y 439.39,Z 376.367,A -85,B 0,C 180,E1 -9199.627,E2 -9199.627} C_VEL
LIN {X 0,Y 439.35,Z 376.376,A -85,B 0,C 180,E1 -9202.577,E2 -9202.577} C_VEL
LIN {X 0,Y 439.358,Z 376.373,A -85,B 0,C 180,E1 -9205.588,E2 -9205.588} C_VEL
LIN {X 0,Y 439.38,Z 376.378,A -85,B 0,C 180,E1 -9208.676,E2 -9208.676} C_VEL
LIN {X 0,Y 439.355,Z 376.37,A -85,B 0,C 180,E1 -9212.03,E2 -9212.03} C_VEL
LIN {X 0,Y 439.383,Z 376.376,A -85,B 0,C 180,E1 -9215.341,E2 -9215.341} C_VEL
LIN {X 0,Y 439.359,Z 376.383,A -85,B 0,C 180,E1 -9218.598,E2 -9218.598} C_VEL
LIN {X 0,Y 439.356,Z 376.38,A -85,B 0,C 180,E1 -9221.254,E2 -9221.254} C_VEL
LIN {X 0,Y 439.391,Z 376.373,A -85,B 0,C 180,E1 -9224.731,E2 -9224.731} C_VEL
LIN {X 0,Y 439.352,Z 376.381,A -85,B 0,C 180,E1 -9227.792,E2 -9227.792} C_VEL
LIN {X 0,Y 439.353,Z 376.379,A -85,B 0,C 180,E1 -9230.221,E2 -9230.221} C_VEL
LIN {X 0,Y 439.367,Z 376.378,A -85,B 0,C 180,E1 -9233.714,E2 -9233.714} C_VEL
LIN {X 0,Y 439.379,Z 376.381,A -85,B 0,C 180,E1 -9235.29,E2 -9235.29} C_VEL
LIN {X 0,Y 440.388,Z 379.203,A -85,B 0,C 180,E1 -9235.421,E2 -9235.421} C_VEL
LIN {X 0,Y 449.655,Z 397.365,A -85,B 0,C 180,E1 -9236.394,E2 -9236.394} C_VEL
LIN {X 0,Y 450.792,Z 399.849,A -85,B 0,C 180,E1 -9236.514,E2 -9236.514} C_VEL
LIN {X 0,Y 449.294,Z 504.4,A -85,B 0,C 180,E1 -9238.268,E2 -9238.268} C_VEL
LIN {X 0,Y 449.044,Z 519.727,A -85,B 0,C 180,E1 -9238.675,E2 -9238.675} C_VEL
LIN {X 0,Y 448.59,Z 533.885,A -85,B 0,C 180,E1 -9239.225,E2 -9239.225} C_VEL
LIN {X 0,Y 447.87,Z 548.591,A -85,B 0,C 180,E1 -9239.989,E2 -9239.989} C_VEL
LIN {X 0,Y 446.958,Z 563.068,A -85,B 0,C 180,E1 -9240.957,E2 -9240.957} C_VEL
LIN {X 0,Y 445.961,Z 576.656,A -85,B 0,C 180,E1 -9242.095,E2 -9242.095} C_VEL
LIN {X 0,Y 445.003,Z 588.027,A -85,B 0,C 180,E1 -9243.251,E2 -9243.251} C_VEL
LIN {X 0,Y 443.88,Z 599.844,A -85,B 0,C 180,E1 -9244.692,E2 -9244.692} C_VEL
LIN {X 0,Y 442.919,Z 609.673,A -85,B 0,C 180,E1 -9246.134,E2 -9246.134} C_VEL
LIN {X 0,Y 442.746,Z 611.132,A -85,B 0,C 180,E1 -9246.368,E2 -9246.368} C_VEL
LIN {X 0,Y 441.706,Z 614.835,A -85,B 0,C 180,E1 -9246.95,E2 -9246.95} C_VEL
LIN {X 0,Y 438.368,Z 620.757,A -85,B 0,C 180,E1 -9247.892,E2 -9247.892} C_VEL
LIN {X 0,Y 435.094,Z 626.271,A -85,B 0,C 180,E1 -9248.888,E2 -9248.888} C_VEL
LIN {X 0,Y 434.166,Z 629.194,A -85,B 0,C 180,E1 -9249.549,E2 -9249.549} C_VEL
LIN {X 0,Y 433.626,Z 634.853,A -85,B 0,C 180,E1 -9251.087,E2 -9251.087} C_VEL
LIN {X 0,Y 433.034,Z 640.576,A -85,B 0,C 180,E1 -9253.015,E2 -9253.015} C_VEL
LIN {X 0,Y 432.598,Z 644.891,A -85,B 0,C 180,E1 -9254.934,E2 -9254.934} C_VEL
LIN {X 0,Y 432.314,Z 647.931,A -85,B 0,C 180,E1 -9256.845,E2 -9256.845} C_VEL
LIN {X 0,Y 432.137,Z 649.761,A -85,B 0,C 180,E1 -9258.747,E2 -9258.747} C_VEL
LIN {X 0,Y 432.141,Z 650.421,A -85,B 0,C 180,E1 -9260.641,E2 -9260.641} C_VEL
LIN {X 0,Y 432.179,Z 649.879,A -85,B 0,C 180,E1 -9262.736,E2 -9262.736} C_VEL
LIN {X 0,Y 432.295,Z 648.457,A -85,B 0,C 180,E1 -9264.403,E2 -9264.403} C_VEL
LIN {X 0,Y 432.35,Z 645.836,A -85,B 0,C 180,E1 -9266.272,E2 -9266.272} C_VEL
LIN {X 0,Y 432.682,Z 642.005,A -85,B 0,C 180,E1 -9268.139,E2 -9268.139} C_VEL
LIN {X 0,Y 433.054,Z 636.904,A -85,B 0,C 180,E1 -9270,E2 -9270} C_VEL
LIN {X 0,Y 433.722,Z 630.387,A -85,B 0,C 180,E1 -9271.857,E2 -9271.857} C_VEL
LIN {X 0,Y 434.429,Z 622.32,A -85,B 0,C 180,E1 -9273.71,E2 -9273.71} C_VEL
LIN {X 0,Y 435.251,Z 613.699,A -85,B 0,C 180,E1 -9275.328,E2 -9275.328} C_VEL
LIN {X 0,Y 436.217,Z 603.362,A -85,B 0,C 180,E1 -9276.94,E2 -9276.94} C_VEL
LIN {X 0,Y 437.096,Z 592.74,A -85,B 0,C 180,E1 -9278.321,E2 -9278.321} C_VEL
LIN {X 0,Y 437.983,Z 581.141,A -85,B 0,C 180,E1 -9279.583,E2 -9279.583} C_VEL
LIN {X 0,Y 439.022,Z 568.401,A -85,B 0,C 180,E1 -9280.725,E2 -9280.725} C_VEL
LIN {X 0,Y 439.813,Z 556.04,A -85,B 0,C 180,E1 -9281.639,E2 -9281.639} C_VEL
LIN {X 0,Y 440.615,Z 541.581,A -85,B 0,C 180,E1 -9282.493,E2 -9282.493} C_VEL
LIN {X 0,Y 441.186,Z 526.365,A -85,B 0,C 180,E1 -9283.179,E2 -9283.179} C_VEL
LIN {X 0,Y 441.485,Z 511.384,A -85,B 0,C 180,E1 -9283.661,E2 -9283.661} C_VEL
LIN {X 0,Y 441.603,Z 492.952,A -85,B 0,C 180,E1 -9284.03,E2 -9284.03} C_VEL
LIN {X 0,Y 442.809,Z 400.837,A -85,B 0,C 180,E1 -9285.558,E2 -9285.558} C_VEL
LIN {X 0,Y 432.564,Z 378.334,A -85,B 0,C 180,E1 -9286.545,E2 -9286.545} C_VEL
LIN {X 0,Y 432.342,Z 377.256,A -85,B 0,C 180,E1 -9286.585,E2 -9286.585} C_VEL
LIN {X 0,Y 432.317,Z 377.257,A -85,B 0,C 180,E1 -9289.961,E2 -9289.961} C_VEL
LIN {X 0,Y 432.299,Z 377.263,A -85,B 0,C 180,E1 -9292.965,E2 -9292.965} C_VEL
LIN {X 0,Y 432.304,Z 377.259,A -85,B 0,C 180,E1 -9296.036,E2 -9296.036} C_VEL
LIN {X 0,Y 432.314,Z 377.251,A -85,B 0,C 180,E1 -9299.189,E2 -9299.189} C_VEL
LIN {X 0,Y 432.304,Z 377.26,A -85,B 0,C 180,E1 -9302.444,E2 -9302.444} C_VEL
LIN {X 0,Y 432.33,Z 377.254,A -85,B 0,C 180,E1 -9305.818,E2 -9305.818} C_VEL
LIN {X 0,Y 432.297,Z 377.259,A -85,B 0,C 180,E1 -9309.348,E2 -9309.348} C_VEL
LIN {X 0,Y 432.299,Z 377.259,A -85,B 0,C 180,E1 -9311.8,E2 -9311.8} C_VEL
LIN {X 0,Y 432.307,Z 377.254,A -85,B 0,C 180,E1 -9314.35,E2 -9314.35} C_VEL
LIN {X 0,Y 432.297,Z 377.261,A -85,B 0,C 180,E1 -9317.018,E2 -9317.018} C_VEL
LIN {X 0,Y 432.284,Z 377.261,A -85,B 0,C 180,E1 -9319.827,E2 -9319.827} C_VEL
LIN {X 0,Y 432.292,Z 377.261,A -85,B 0,C 180,E1 -9323.02,E2 -9323.02} C_VEL
LIN {X 0,Y 432.325,Z 377.25,A -85,B 0,C 180,E1 -9326.002,E2 -9326.002} C_VEL
LIN {X 0,Y 432.324,Z 377.257,A -85,B 0,C 180,E1 -9329.493,E2 -9329.493} C_VEL
LIN {X 0,Y 432.305,Z 377.258,A -85,B 0,C 180,E1 -9331.871,E2 -9331.871} C_VEL
LIN {X 0,Y 432.34,Z 377.251,A -85,B 0,C 180,E1 -9335.547,E2 -9335.547} C_VEL
LIN {X 0,Y 432.342,Z 377.256,A -85,B 0,C 180,E1 -9339.045,E2 -9339.045} C_VEL
LIN {X 0,Y 432.349,Z 377.25,A -85,B 0,C 180,E1 -9342.01,E2 -9342.01} C_VEL
LIN {X 0,Y 432.371,Z 377.25,A -85,B 0,C 180,E1 -9344.925,E2 -9344.925} C_VEL
LIN {X 0,Y 432.45,Z 377.219,A -85,B 0,C 180,E1 -9347.803,E2 -9347.803} C_VEL
LIN {X 0,Y 432.437,Z 377.232,A -85,B 0,C 180,E1 -9351.589,E2 -9351.589} C_VEL
LIN {X 0,Y 432.541,Z 377.227,A -85,B 0,C 180,E1 -9354.405,E2 -9354.405} C_VEL
LIN {X 0,Y 432.581,Z 377.217,A -85,B 0,C 180,E1 -9358.138,E2 -9358.138} C_VEL
LIN {X 0,Y 432.455,Z 377.238,A -85,B 0,C 180,E1 -9360.931,E2 -9360.931} C_VEL
LIN {X 0,Y 432.555,Z 377.222,A -85,B 0,C 180,E1 -9362.794,E2 -9362.794} C_VEL
LIN {X 0,Y 432.5,Z 377.232,A -85,B 0,C 180,E1 -9366.531,E2 -9366.531} C_VEL
LIN {X 0,Y 432.414,Z 377.241,A -85,B 0,C 180,E1 -9369.354,E2 -9369.354} C_VEL
LIN {X 0,Y 432.422,Z 377.242,A -85,B 0,C 180,E1 -9372.803,E2 -9372.803} C_VEL
LIN {X 0,Y 432.347,Z 377.252,A -85,B 0,C 180,E1 -9376.453,E2 -9376.453} C_VEL
LIN {X 0,Y 432.304,Z 377.262,A -85,B 0,C 180,E1 -9379.962,E2 -9379.962} C_VEL
LIN {X 0,Y 432.294,Z 377.255,A -85,B 0,C 180,E1 -9382.965,E2 -9382.965} C_VEL
LIN {X 0,Y 432.309,Z 377.257,A -85,B 0,C 180,E1 -9386.036,E2 -9386.036} C_VEL
LIN {X 0,Y 432.314,Z 377.257,A -85,B 0,C 180,E1 -9389.189,E2 -9389.189} C_VEL
LIN {X 0,Y 432.311,Z 377.254,A -85,B 0,C 180,E1 -9392.444,E2 -9392.444} C_VEL
LIN {X 0,Y 432.325,Z 377.261,A -85,B 0,C 180,E1 -9395.819,E2 -9395.819} C_VEL
LIN {X 0,Y 432.293,Z 377.255,A -85,B 0,C 180,E1 -9399.349,E2 -9399.349} C_VEL
LIN {X 0,Y 432.296,Z 377.258,A -85,B 0,C 180,E1 -9401.801,E2 -9401.801} C_VEL
LIN {X 0,Y 432.326,Z 377.257,A -85,B 0,C 180,E1 -9404.348,E2 -9404.348} C_VEL
LIN {X 0,Y 432.296,Z 377.261,A -85,B 0,C 180,E1 -9407.019,E2 -9407.019} C_VEL
LIN {X 0,Y 432.282,Z 377.245,A -85,B 0,C 180,E1 -9409.829,E2 -9409.829} C_VEL
LIN {X 0,Y 432.291,Z 377.262,A -85,B 0,C 180,E1 -9413.021,E2 -9413.021} C_VEL
LIN {X 0,Y 432.355,Z 377.381,A -85,B 0,C 180,E1 -9413.591,E2 -9413.591} C_VEL
LIN {X 0,Y 437.241,Z 395.385,A -85,B 0,C 180,E1 -9416.292,E2 -9416.292} C_VEL
LIN {X 0,Y 439.857,Z 406.437,A -85,B 0,C 180,E1 -9417.868,E2 -9417.868} C_VEL
LIN {X 0,Y 438.266,Z 431.749,A -85,B 0,C 180,E1 -9420.982,E2 -9420.982} C_VEL
LIN {X 0,Y 436.76,Z 456.779,A -85,B 0,C 180,E1 -9424.025,E2 -9424.025} C_VEL
LIN {X 0,Y 442.389,Z 496.905,A -85,B 0,C 180,E1 -9425.034,E2 -9425.034} C_VEL
LIN {X 0,Y 440.545,Z 626.217,A -85,B 0,C 180,E1 -9427.179,E2 -9427.179} C_VEL
LIN {X 0,Y 439.822,Z 642.084,A -85,B 0,C 180,E1 -9427.62,E2 -9427.62} C_VEL
LIN {X 0,Y 438.901,Z 656.36,A -85,B 0,C 180,E1 -9428.19,E2 -9428.19} C_VEL
LIN {X 0,Y 437.871,Z 670.807,A -85,B 0,C 180,E1 -9428.954,E2 -9428.954} C_VEL
LIN {X 0,Y 436.77,Z 684.676,A -85,B 0,C 180,E1 -9429.883,E2 -9429.883} C_VEL
LIN {X 0,Y 435.697,Z 697.469,A -85,B 0,C 180,E1 -9430.935,E2 -9430.935} C_VEL
LIN {X 0,Y 434.747,Z 709.4,A -85,B 0,C 180,E1 -9432.113,E2 -9432.113} C_VEL
LIN {X 0,Y 433.762,Z 721.432,A -85,B 0,C 180,E1 -9433.528,E2 -9433.528} C_VEL
LIN {X 0,Y 432.968,Z 731.573,A -85,B 0,C 180,E1 -9434.947,E2 -9434.947} C_VEL
LIN {X 0,Y 432.369,Z 741.549,A -85,B 0,C 180,E1 -9436.607,E2 -9436.607} C_VEL
LIN {X 0,Y 431.947,Z 749.877,A -85,B 0,C 180,E1 -9438.265,E2 -9438.265} C_VEL
LIN {X 0,Y 431.763,Z 755.88,A -85,B 0,C 180,E1 -9439.685,E2 -9439.685} C_VEL
LIN {X 0,Y 431.664,Z 762.451,A -85,B 0,C 180,E1 -9441.574,E2 -9441.574} C_VEL
LIN {X 0,Y 431.697,Z 767.549,A -85,B 0,C 180,E1 -9443.456,E2 -9443.456} C_VEL
LIN {X 0,Y 431.764,Z 771.287,A -85,B 0,C 180,E1 -9445.331,E2 -9445.331} C_VEL
LIN {X 0,Y 431.769,Z 773.739,A -85,B 0,C 180,E1 -9447.201,E2 -9447.201} C_VEL
LIN {X 0,Y 431.938,Z 774.996,A -85,B 0,C 180,E1 -9449.067,E2 -9449.067} C_VEL
LIN {X 0,Y 431.939,Z 774.981,A -85,B 0,C 180,E1 -9450.932,E2 -9450.932} C_VEL
LIN {X 0,Y 431.77,Z 773.73,A -85,B 0,C 180,E1 -9452.799,E2 -9452.799} C_VEL
LIN {X 0,Y 431.782,Z 771.301,A -85,B 0,C 180,E1 -9454.668,E2 -9454.668} C_VEL
LIN {X 0,Y 431.705,Z 767.094,A -85,B 0,C 180,E1 -9456.756,E2 -9456.756} C_VEL
LIN {X 0,Y 431.645,Z 762.577,A -85,B 0,C 180,E1 -9458.426,E2 -9458.426} C_VEL
LIN {X 0,Y 431.758,Z 756.105,A -85,B 0,C 180,E1 -9460.314,E2 -9460.314} C_VEL
LIN {X 0,Y 431.995,Z 748.021,A -85,B 0,C 180,E1 -9462.209,E2 -9462.209} C_VEL
LIN {X 0,Y 432.533,Z 739.482,A -85,B 0,C 180,E1 -9463.866,E2 -9463.866} C_VEL
LIN {X 0,Y 433.25,Z 729.268,A -85,B 0,C 180,E1 -9465.524,E2 -9465.524} C_VEL
LIN {X 0,Y 434.288,Z 717.066,A -85,B 0,C 180,E1 -9467.169,E2 -9467.169} C_VEL
LIN {X 0,Y 435.384,Z 704.337,A -85,B 0,C 180,E1 -9468.59,E2 -9468.59} C_VEL
LIN {X 0,Y 436.503,Z 691.741,A -85,B 0,C 180,E1 -9469.761,E2 -9469.761} C_VEL
LIN {X 0,Y 437.764,Z 678.036,A -85,B 0,C 180,E1 -9470.805,E2 -9470.805} C_VEL
LIN {X 0,Y 438.933,Z 663.559,A -85,B 0,C 180,E1 -9471.691,E2 -9471.691} C_VEL
LIN {X 0,Y 440.115,Z 648.142,A -85,B 0,C 180,E1 -9472.411,E2 -9472.411} C_VEL
LIN {X 0,Y 441.026,Z 633.126,A -85,B 0,C 180,E1 -9472.918,E2 -9472.918} C_VEL
LIN {X 0,Y 441.612,Z 617.668,A -85,B 0,C 180,E1 -9473.257,E2 -9473.257} C_VEL
LIN {X 0,Y 443.41,Z 497.036,A -85,B 0,C 180,E1 -9475.277,E2 -9475.277} C_VEL
LIN {X 0,Y 439.081,Z 465.707,A -85,B 0,C 180,E1 -9476.124,E2 -9476.124} C_VEL
LIN {X 0,Y 437.389,Z 455.423,A -85,B 0,C 180,E1 -9476.454,E2 -9476.454} C_VEL
LIN {X 0,Y 439.202,Z 429.214,A -85,B 0,C 180,E1 -9479.738,E2 -9479.738} C_VEL
LIN {X 0,Y 440.737,Z 408.994,A -85,B 0,C 180,E1 -9482.314,E2 -9482.314} C_VEL
LIN {X 0,Y 440.52,Z 406.426,A -85,B 0,C 180,E1 -9482.672,E2 -9482.672} C_VEL
LIN {X 0,Y 436.325,Z 390.408,A -85,B 0,C 180,E1 -9485.183,E2 -9485.183} C_VEL
LIN {X 0,Y 432.294,Z 377.262,A -85,B 0,C 180,E1 -9487.435,E2 -9487.435} C_VEL
LIN {X 0,Y 432.281,Z 377.263,A -85,B 0,C 180,E1 -9490.564,E2 -9490.564} C_VEL
LIN {X 0,Y 432.295,Z 377.259,A -85,B 0,C 180,E1 -9493.062,E2 -9493.062} C_VEL
LIN {X 0,Y 432.322,Z 377.242,A -85,B 0,C 180,E1 -9495.664,E2 -9495.664} C_VEL
LIN {X 0,Y 432.296,Z 377.259,A -85,B 0,C 180,E1 -9498.401,E2 -9498.401} C_VEL
LIN {X 0,Y 432.31,Z 377.256,A -85,B 0,C 180,E1 -9501.847,E2 -9501.847} C_VEL
LIN {X 0,Y 432.313,Z 377.258,A -85,B 0,C 180,E1 -9505.321,E2 -9505.321} C_VEL
LIN {X 0,Y 432.304,Z 377.259,A -85,B 0,C 180,E1 -9508.653,E2 -9508.653} C_VEL
LIN {X 0,Y 432.307,Z 377.262,A -85,B 0,C 180,E1 -9511.872,E2 -9511.872} C_VEL
LIN {X 0,Y 432.309,Z 377.257,A -85,B 0,C 180,E1 -9514.996,E2 -9514.996} C_VEL
LIN {X 0,Y 432.337,Z 377.259,A -85,B 0,C 180,E1 -9518.045,E2 -9518.045} C_VEL
LIN {X 0,Y 432.329,Z 377.257,A -85,B 0,C 180,E1 -9521.027,E2 -9521.027} C_VEL
LIN {X 0,Y 432.37,Z 377.251,A -85,B 0,C 180,E1 -9523.959,E2 -9523.959} C_VEL
LIN {X 0,Y 432.444,Z 377.241,A -85,B 0,C 180,E1 -9527.803,E2 -9527.803} C_VEL
LIN {X 0,Y 432.432,Z 377.242,A -85,B 0,C 180,E1 -9531.589,E2 -9531.589} C_VEL
LIN {X 0,Y 432.531,Z 377.229,A -85,B 0,C 180,E1 -9534.405,E2 -9534.405} C_VEL
LIN {X 0,Y 432.584,Z 377.22,A -85,B 0,C 180,E1 -9538.138,E2 -9538.138} C_VEL
LIN {X 0,Y 432.541,Z 377.226,A -85,B 0,C 180,E1 -9540.931,E2 -9540.931} C_VEL
LIN {X 0,Y 432.548,Z 377.232,A -85,B 0,C 180,E1 -9542.794,E2 -9542.794} C_VEL
LIN {X 0,Y 432.569,Z 377.214,A -85,B 0,C 180,E1 -9545.594,E2 -9545.594} C_VEL
LIN {X 0,Y 432.437,Z 377.228,A -85,B 0,C 180,E1 -9548.411,E2 -9548.411} C_VEL
LIN {X 0,Y 432.445,Z 377.241,A -85,B 0,C 180,E1 -9552.197,E2 -9552.197} C_VEL
LIN {X 0,Y 432.417,Z 377.237,A -85,B 0,C 180,E1 -9556.04,E2 -9556.04} C_VEL
LIN {X 0,Y 432.375,Z 377.241,A -85,B 0,C 180,E1 -9559.486,E2 -9559.486} C_VEL
LIN {X 0,Y 432.298,Z 377.261,A -85,B 0,C 180,E1 -9562.966,E2 -9562.966} C_VEL
LIN {X 0,Y 432.308,Z 377.251,A -85,B 0,C 180,E1 -9566.036,E2 -9566.036} C_VEL
LIN {X 0,Y 432.316,Z 377.262,A -85,B 0,C 180,E1 -9569.19,E2 -9569.19} C_VEL
LIN {X 0,Y 432.311,Z 377.249,A -85,B 0,C 180,E1 -9572.444,E2 -9572.444} C_VEL
LIN {X 0,Y 432.328,Z 377.253,A -85,B 0,C 180,E1 -9575.819,E2 -9575.819} C_VEL
LIN {X 0,Y 432.322,Z 377.261,A -85,B 0,C 180,E1 -9578.714,E2 -9578.714} C_VEL
LIN {X 0,Y 432.297,Z 377.259,A -85,B 0,C 180,E1 -9581.802,E2 -9581.802} C_VEL
LIN {X 0,Y 432.327,Z 377.249,A -85,B 0,C 180,E1 -9584.349,E2 -9584.349} C_VEL
LIN {X 0,Y 432.301,Z 377.257,A -85,B 0,C 180,E1 -9587.019,E2 -9587.019} C_VEL
LIN {X 0,Y 432.303,Z 377.256,A -85,B 0,C 180,E1 -9589.826,E2 -9589.826} C_VEL
LIN {X 0,Y 432.3,Z 377.263,A -85,B 0,C 180,E1 -9593.023,E2 -9593.023} C_VEL
LIN {X 0,Y 432.38,Z 377.425,A -85,B 0,C 180,E1 -9594.796,E2 -9594.796} C_VEL
LIN {X 0,Y 433.424,Z 380.205,A -85,B 0,C 180,E1 -9594.927,E2 -9594.927} C_VEL
LIN {X 0,Y 441.895,Z 396.536,A -85,B 0,C 180,E1 -9595.845,E2 -9595.845} C_VEL
LIN {X 0,Y 444.524,Z 402.005,A -85,B 0,C 180,E1 -9596.128,E2 -9596.128} C_VEL
LIN {X 0,Y 442.923,Z 504.162,A -85,B 0,C 180,E1 -9597.857,E2 -9597.857} C_VEL
LIN {X 0,Y 442.674,Z 519.996,A -85,B 0,C 180,E1 -9598.272,E2 -9598.272} C_VEL
LIN {X 0,Y 442.199,Z 534.466,A -85,B 0,C 180,E1 -9598.835,E2 -9598.835} C_VEL
LIN {X 0,Y 441.477,Z 548.701,A -85,B 0,C 180,E1 -9599.575,E2 -9599.575} C_VEL
LIN {X 0,Y 440.631,Z 562.56,A -85,B 0,C 180,E1 -9600.499,E2 -9600.499} C_VEL
LIN {X 0,Y 439.718,Z 574.428,A -85,B 0,C 180,E1 -9601.465,E2 -9601.465} C_VEL
LIN {X 0,Y 438.594,Z 586.936,A -85,B 0,C 180,E1 -9602.699,E2 -9602.699} C_VEL
LIN {X 0,Y 437.445,Z 598.784,A -85,B 0,C 180,E1 -9604.119,E2 -9604.119} C_VEL
LIN {X 0,Y 436.461,Z 608.471,A -85,B 0,C 180,E1 -9605.505,E2 -9605.505} C_VEL
LIN {X 0,Y 435.393,Z 618.387,A -85,B 0,C 180,E1 -9607.208,E2 -9607.208} C_VEL
LIN {X 0,Y 434.453,Z 626.535,A -85,B 0,C 180,E1 -9608.905,E2 -9608.905} C_VEL
LIN {X 0,Y 434.166,Z 629.194,A -85,B 0,C 180,E1 -9609.549,E2 -9609.549} C_VEL
LIN {X 0,Y 433.254,Z 632.014,A -85,B 0,C 180,E1 -9610.225,E2 -9610.225} C_VEL
LIN {X 0,Y 430.057,Z 636.492,A -85,B 0,C 180,E1 -9611.321,E2 -9611.321} C_VEL
LIN {X 0,Y 426.871,Z 640.46,A -85,B 0,C 180,E1 -9612.462,E2 -9612.462} C_VEL
LIN {X 0,Y 425.993,Z 642.459,A -85,B 0,C 180,E1 -9613.2,E2 -9613.2} C_VEL
LIN {X 0,Y 425.66,Z 645.702,A -85,B 0,C 180,E1 -9614.683,E2 -9614.683} C_VEL
LIN {X 0,Y 425.334,Z 648.805,A -85,B 0,C 180,E1 -9616.625,E2 -9616.625} C_VEL
LIN {X 0,Y 425.129,Z 650.687,A -85,B 0,C 180,E1 -9618.559,E2 -9618.559} C_VEL
LIN {X 0,Y 425.105,Z 651.424,A -85,B 0,C 180,E1 -9620.485,E2 -9620.485} C_VEL
LIN {X 0,Y 425.154,Z 650.923,A -85,B 0,C 180,E1 -9622.673,E2 -9622.673} C_VEL
LIN {X 0,Y 425.286,Z 649.602,A -85,B 0,C 180,E1 -9624.31,E2 -9624.31} C_VEL
LIN {X 0,Y 425.319,Z 647.06,A -85,B 0,C 180,E1 -9626.211,E2 -9626.211} C_VEL
LIN {X 0,Y 425.672,Z 643.273,A -85,B 0,C 180,E1 -9628.108,E2 -9628.108} C_VEL
LIN {X 0,Y 426.048,Z 638.247,A -85,B 0,C 180,E1 -9630,E2 -9630} C_VEL
LIN {X 0,Y 426.747,Z 631.815,A -85,B 0,C 180,E1 -9631.888,E2 -9631.888} C_VEL
LIN {X 0,Y 427.362,Z 624.92,A -85,B 0,C 180,E1 -9633.536,E2 -9633.536} C_VEL
LIN {X 0,Y 428.174,Z 616.639,A -85,B 0,C 180,E1 -9635.18,E2 -9635.18} C_VEL
LIN {X 0,Y 429.209,Z 606.675,A -85,B 0,C 180,E1 -9636.818,E2 -9636.818} C_VEL
LIN {X 0,Y 430.112,Z 596.512,A -85,B 0,C 180,E1 -9638.22,E2 -9638.22} C_VEL
LIN {X 0,Y 431.074,Z 584.352,A -85,B 0,C 180,E1 -9639.62,E2 -9639.62} C_VEL
LIN {X 0,Y 432.084,Z 572.102,A -85,B 0,C 180,E1 -9640.781,E2 -9640.781} C_VEL
LIN {X 0,Y 433.044,Z 558.663,A -85,B 0,C 180,E1 -9641.823,E2 -9641.823} C_VEL
LIN {X 0,Y 433.893,Z 544.646,A -85,B 0,C 180,E1 -9642.69,E2 -9642.69} C_VEL
LIN {X 0,Y 434.529,Z 529.995,A -85,B 0,C 180,E1 -9643.391,E2 -9643.391} C_VEL
LIN {X 0,Y 434.823,Z 515.726,A -85,B 0,C 180,E1 -9643.897,E2 -9643.897} C_VEL
LIN {X 0,Y 434.979,Z 500.468,A -85,B 0,C 180,E1 -9644.248,E2 -9644.248} C_VEL
LIN {X 0,Y 436.29,Z 402.812,A -85,B 0,C 180,E1 -9645.893,E2 -9645.893} C_VEL
LIN {X 0,Y 425.333,Z 378.552,A -85,B 0,C 180,E1 -9646.978,E2 -9646.978} C_VEL
LIN {X 0,Y 425.28,Z 378.132,A -85,B 0,C 180,E1 -9647.021,E2 -9647.021} C_VEL
LIN {X 0,Y 425.28,Z 378.134,A -85,B 0,C 180,E1 -9650.306,E2 -9650.306} C_VEL
LIN {X 0,Y 425.26,Z 378.14,A -85,B 0,C 180,E1 -9653.368,E2 -9653.368} C_VEL
LIN {X 0,Y 425.261,Z 378.138,A -85,B 0,C 180,E1 -9656.5,E2 -9656.5} C_VEL
LIN {X 0,Y 425.27,Z 378.123,A -85,B 0,C 180,E1 -9659.721,E2 -9659.721} C_VEL
LIN {X 0,Y 425.259,Z 378.14,A -85,B 0,C 180,E1 -9663.049,E2 -9663.049} C_VEL
LIN {X 0,Y 425.274,Z 378.133,A -85,B 0,C 180,E1 -9665.926,E2 -9665.926} C_VEL
LIN {X 0,Y 425.254,Z 378.14,A -85,B 0,C 180,E1 -9669.036,E2 -9669.036} C_VEL
LIN {X 0,Y 425.24,Z 378.137,A -85,B 0,C 180,E1 -9671.95,E2 -9671.95} C_VEL
LIN {X 0,Y 425.275,Z 378.139,A -85,B 0,C 180,E1 -9675.283,E2 -9675.283} C_VEL
LIN {X 0,Y 425.243,Z 378.136,A -85,B 0,C 180,E1 -9678.617,E2 -9678.617} C_VEL
LIN {X 0,Y 425.271,Z 378.136,A -85,B 0,C 180,E1 -9681.098,E2 -9681.098} C_VEL
LIN {X 0,Y 425.287,Z 378.133,A -85,B 0,C 180,E1 -9684.663,E2 -9684.663} C_VEL
LIN {X 0,Y 425.239,Z 378.138,A -85,B 0,C 180,E1 -9688.071,E2 -9688.071} C_VEL
LIN {X 0,Y 425.285,Z 378.132,A -85,B 0,C 180,E1 -9691.364,E2 -9691.364} C_VEL
LIN {X 0,Y 425.244,Z 378.137,A -85,B 0,C 180,E1 -9694.551,E2 -9694.551} C_VEL
LIN {X 0,Y 425.285,Z 378.135,A -85,B 0,C 180,E1 -9697.729,E2 -9697.729} C_VEL
LIN {X 0,Y 425.354,Z 378.12,A -85,B 0,C 180,E1 -9700.703,E2 -9700.703} C_VEL
LIN {X 0,Y 425.376,Z 378.124,A -85,B 0,C 180,E1 -9703.688,E2 -9703.688} C_VEL
LIN {X 0,Y 425.403,Z 378.099,A -85,B 0,C 180,E1 -9707.598,E2 -9707.598} C_VEL
LIN {X 0,Y 425.386,Z 378.107,A -85,B 0,C 180,E1 -9711.449,E2 -9711.449} C_VEL
LIN {X 0,Y 425.499,Z 378.105,A -85,B 0,C 180,E1 -9714.312,E2 -9714.312} C_VEL
LIN {X 0,Y 425.55,Z 378.093,A -85,B 0,C 180,E1 -9718.107,E2 -9718.107} C_VEL
LIN {X 0,Y 425.425,Z 378.114,A -85,B 0,C 180,E1 -9720.946,E2 -9720.946} C_VEL
LIN {X 0,Y 425.511,Z 378.1,A -85,B 0,C 180,E1 -9722.84,E2 -9722.84} C_VEL
LIN {X 0,Y 425.462,Z 378.108,A -85,B 0,C 180,E1 -9726.64,E2 -9726.64} C_VEL
LIN {X 0,Y 425.375,Z 378.118,A -85,B 0,C 180,E1 -9729.51,E2 -9729.51} C_VEL
LIN {X 0,Y 425.385,Z 378.119,A -85,B 0,C 180,E1 -9732.903,E2 -9732.903} C_VEL
LIN {X 0,Y 425.304,Z 378.13,A -85,B 0,C 180,E1 -9736.583,E2 -9736.583} C_VEL
LIN {X 0,Y 425.287,Z 378.133,A -85,B 0,C 180,E1 -9739.623,E2 -9739.623} C_VEL
LIN {X 0,Y 425.276,Z 378.13,A -85,B 0,C 180,E1 -9742.339,E2 -9742.339} C_VEL
LIN {X 0,Y 425.251,Z 378.14,A -85,B 0,C 180,E1 -9745.448,E2 -9745.448} C_VEL
LIN {X 0,Y 425.292,Z 378.13,A -85,B 0,C 180,E1 -9748.859,E2 -9748.859} C_VEL
LIN {X 0,Y 425.253,Z 378.138,A -85,B 0,C 180,E1 -9751.928,E2 -9751.928} C_VEL
LIN {X 0,Y 425.285,Z 378.132,A -85,B 0,C 180,E1 -9755.337,E2 -9755.337} C_VEL
LIN {X 0,Y 425.268,Z 378.127,A -85,B 0,C 180,E1 -9758.902,E2 -9758.902} C_VEL
LIN {X 0,Y 425.249,Z 378.133,A -85,B 0,C 180,E1 -9762.656,E2 -9762.656} C_VEL
LIN {X 0,Y 425.278,Z 378.133,A -85,B 0,C 180,E1 -9765.284,E2 -9765.284} C_VEL
LIN {X 0,Y 425.24,Z 378.128,A -85,B 0,C 180,E1 -9768.618,E2 -9768.618} C_VEL
LIN {X 0,Y 425.264,Z 378.14,A -85,B 0,C 180,E1 -9772.305,E2 -9772.305} C_VEL
LIN {X 0,Y 425.284,Z 378.257,A -85,B 0,C 180,E1 -9773.219,E2 -9773.219} C_VEL
LIN {X 0,Y 430.329,Z 396.719,A -85,B 0,C 180,E1 -9776.048,E2 -9776.048} C_VEL
LIN {X 0,Y 432.966,Z 407.449,A -85,B 0,C 180,E1 -9777.612,E2 -9777.612} C_VEL
LIN {X 0,Y 431.885,Z 425.186,A -85,B 0,C 180,E1 -9779.84,E2 -9779.84} C_VEL
LIN {X 0,Y 430.402,Z 448.98,A -85,B 0,C 180,E1 -9782.793,E2 -9782.793} C_VEL
LIN {X 0,Y 429.939,Z 455.806,A -85,B 0,C 180,E1 -9783.633,E2 -9783.633} C_VEL
LIN {X 0,Y 435.763,Z 497.269,A -85,B 0,C 180,E1 -9784.691,E2 -9784.691} C_VEL
LIN {X 0,Y 434.103,Z 613.73,A -85,B 0,C 180,E1 -9786.632,E2 -9786.632} C_VEL
LIN {X 0,Y 433.643,Z 630.845,A -85,B 0,C 180,E1 -9786.984,E2 -9786.984} C_VEL
LIN {X 0,Y 432.836,Z 645.995,A -85,B 0,C 180,E1 -9787.475,E2 -9787.475} C_VEL
LIN {X 0,Y 431.848,Z 660.209,A -85,B 0,C 180,E1 -9788.111,E2 -9788.111} C_VEL
LIN {X 0,Y 430.716,Z 674.812,A -85,B 0,C 180,E1 -9788.963,E2 -9788.963} C_VEL
LIN {X 0,Y 429.477,Z 689.229,A -85,B 0,C 180,E1 -9790.026,E2 -9790.026} C_VEL
LIN {X 0,Y 428.371,Z 702.353,A -85,B 0,C 180,E1 -9791.218,E2 -9791.218} C_VEL
LIN {X 0,Y 427.339,Z 714.357,A -85,B 0,C 180,E1 -9792.528,E2 -9792.528} C_VEL
LIN {X 0,Y 426.41,Z 725.478,A -85,B 0,C 180,E1 -9793.974,E2 -9793.974} C_VEL
LIN {X 0,Y 425.623,Z 736.301,A -85,B 0,C 180,E1 -9795.659,E2 -9795.659} C_VEL
LIN {X 0,Y 425.073,Z 745.036,A -85,B 0,C 180,E1 -9797.286,E2 -9797.286} C_VEL
LIN {X 0,Y 424.822,Z 752.867,A -85,B 0,C 180,E1 -9799.033,E2 -9799.033} C_VEL
LIN {X 0,Y 424.584,Z 759.85,A -85,B 0,C 180,E1 -9800.953,E2 -9800.953} C_VEL
LIN {X 0,Y 424.609,Z 765.348,A -85,B 0,C 180,E1 -9802.869,E2 -9802.869} C_VEL
LIN {X 0,Y 424.643,Z 768.514,A -85,B 0,C 180,E1 -9804.301,E2 -9804.301} C_VEL
LIN {X 0,Y 424.724,Z 771.626,A -85,B 0,C 180,E1 -9806.205,E2 -9806.205} C_VEL
LIN {X 0,Y 424.738,Z 773.48,A -85,B 0,C 180,E1 -9808.103,E2 -9808.103} C_VEL
LIN {X 0,Y 424.917,Z 773.978,A -85,B 0,C 180,E1 -9809.052,E2 -9809.052} C_VEL
LIN {X 0,Y 424.917,Z 773.968,A -85,B 0,C 180,E1 -9810.947,E2 -9810.947} C_VEL
LIN {X 0,Y 424.729,Z 772.728,A -85,B 0,C 180,E1 -9812.845,E2 -9812.845} C_VEL
LIN {X 0,Y 424.728,Z 770.309,A -85,B 0,C 180,E1 -9814.745,E2 -9814.745} C_VEL
LIN {X 0,Y 424.652,Z 766.317,A -85,B 0,C 180,E1 -9816.784,E2 -9816.784} C_VEL
LIN {X 0,Y 424.58,Z 761.612,A -85,B 0,C 180,E1 -9818.567,E2 -9818.567} C_VEL
LIN {X 0,Y 424.706,Z 755.159,A -85,B 0,C 180,E1 -9820.487,E2 -9820.487} C_VEL
LIN {X 0,Y 424.949,Z 747.098,A -85,B 0,C 180,E1 -9822.415,E2 -9822.415} C_VEL
LIN {X 0,Y 425.522,Z 738.576,A -85,B 0,C 180,E1 -9824.099,E2 -9824.099} C_VEL
LIN {X 0,Y 426.306,Z 728.4,A -85,B 0,C 180,E1 -9825.783,E2 -9825.783} C_VEL
LIN {X 0,Y 427.306,Z 717.232,A -85,B 0,C 180,E1 -9827.33,E2 -9827.33} C_VEL
LIN {X 0,Y 428.449,Z 704.737,A -85,B 0,C 180,E1 -9828.778,E2 -9828.778} C_VEL
LIN {X 0,Y 429.624,Z 692.385,A -85,B 0,C 180,E1 -9829.966,E2 -9829.966} C_VEL
LIN {X 0,Y 430.907,Z 679.047,A -85,B 0,C 180,E1 -9831.026,E2 -9831.026} C_VEL
LIN {X 0,Y 432.213,Z 664.447,A -85,B 0,C 180,E1 -9831.961,E2 -9831.961} C_VEL
LIN {X 0,Y 433.392,Z 649.617,A -85,B 0,C 180,E1 -9832.695,E2 -9832.695} C_VEL
LIN {X 0,Y 434.455,Z 634.096,A -85,B 0,C 180,E1 -9833.253,E2 -9833.253} C_VEL
LIN {X 0,Y 435.068,Z 619.914,A -85,B 0,C 180,E1 -9833.597,E2 -9833.597} C_VEL
LIN {X 0,Y 437.079,Z 498.205,A -85,B 0,C 180,E1 -9835.669,E2 -9835.669} C_VEL
LIN {X 0,Y 433.005,Z 468.214,A -85,B 0,C 180,E1 -9836.495,E2 -9836.495} C_VEL
LIN {X 0,Y 430.732,Z 454.411,A -85,B 0,C 180,E1 -9836.928,E2 -9836.928} C_VEL
LIN {X 0,Y 432.608,Z 428.508,A -85,B 0,C 180,E1 -9840.238,E2 -9840.238} C_VEL
LIN {X 0,Y 434.134,Z 409.767,A -85,B 0,C 180,E1 -9842.669,E2 -9842.669} C_VEL
LIN {X 0,Y 430.056,Z 393.792,A -85,B 0,C 180,E1 -9845.204,E2 -9845.204} C_VEL
LIN {X 0,Y 425.251,Z 378.139,A -85,B 0,C 180,E1 -9847.92,E2 -9847.92} C_VEL
LIN {X 0,Y 425.24,Z 378.138,A -85,B 0,C 180,E1 -9851.381,E2 -9851.381} C_VEL
LIN {X 0,Y 425.274,Z 378.125,A -85,B 0,C 180,E1 -9854.716,E2 -9854.716} C_VEL
LIN {X 0,Y 425.254,Z 378.139,A -85,B 0,C 180,E1 -9858.045,E2 -9858.045} C_VEL
LIN {X 0,Y 425.265,Z 378.131,A -85,B 0,C 180,E1 -9861.098,E2 -9861.098} C_VEL
LIN {X 0,Y 425.28,Z 378.137,A -85,B 0,C 180,E1 -9864.662,E2 -9864.662} C_VEL
LIN {X 0,Y 425.249,Z 378.142,A -85,B 0,C 180,E1 -9868.072,E2 -9868.072} C_VEL
LIN {X 0,Y 425.283,Z 378.134,A -85,B 0,C 180,E1 -9871.365,E2 -9871.365} C_VEL
LIN {X 0,Y 425.246,Z 378.141,A -85,B 0,C 180,E1 -9874.552,E2 -9874.552} C_VEL
LIN {X 0,Y 425.276,Z 378.136,A -85,B 0,C 180,E1 -9877.73,E2 -9877.73} C_VEL
LIN {X 0,Y 425.309,Z 378.134,A -85,B 0,C 180,E1 -9880.702,E2 -9880.702} C_VEL
LIN {X 0,Y 425.304,Z 378.13,A -85,B 0,C 180,E1 -9883.685,E2 -9883.685} C_VEL
LIN {X 0,Y 425.397,Z 378.118,A -85,B 0,C 180,E1 -9887.598,E2 -9887.598} C_VEL
LIN {X 0,Y 425.381,Z 378.12,A -85,B 0,C 180,E1 -9891.449,E2 -9891.449} C_VEL
LIN {X 0,Y 425.488,Z 378.105,A -85,B 0,C 180,E1 -9894.313,E2 -9894.313} C_VEL
LIN {X 0,Y 425.553,Z 378.095,A -85,B 0,C 180,E1 -9898.107,E2 -9898.107} C_VEL
LIN {X 0,Y 425.503,Z 378.102,A -85,B 0,C 180,E1 -9900.947,E2 -9900.947} C_VEL
LIN {X 0,Y 425.504,Z 378.109,A -85,B 0,C 180,E1 -9902.84,E2 -9902.84} C_VEL
LIN {X 0,Y 425.525,Z 378.091,A -85,B 0,C 180,E1 -9905.687,E2 -9905.687} C_VEL
LIN {X 0,Y 425.385,Z 378.108,A -85,B 0,C 180,E1 -9908.551,E2 -9908.551} C_VEL
LIN {X 0,Y 425.398,Z 378.117,A -85,B 0,C 180,E1 -9912.402,E2 -9912.402} C_VEL
LIN {X 0,Y 425.375,Z 378.116,A -85,B 0,C 180,E1 -9916.313,E2 -9916.313} C_VEL
LIN {X 0,Y 425.316,Z 378.12,A -85,B 0,C 180,E1 -9919.636,E2 -9919.636} C_VEL
LIN {X 0,Y 425.275,Z 378.126,A -85,B 0,C 180,E1 -9922.34,E2 -9922.34} C_VEL
LIN {X 0,Y 425.25,Z 378.131,A -85,B 0,C 180,E1 -9925.449,E2 -9925.449} C_VEL
LIN {X 0,Y 425.297,Z 378.134,A -85,B 0,C 180,E1 -9928.861,E2 -9928.861} C_VEL
LIN {X 0,Y 425.252,Z 378.126,A -85,B 0,C 180,E1 -9931.928,E2 -9931.928} C_VEL
LIN {X 0,Y 425.287,Z 378.132,A -85,B 0,C 180,E1 -9935.338,E2 -9935.338} C_VEL
LIN {X 0,Y 425.276,Z 378.14,A -85,B 0,C 180,E1 -9938.902,E2 -9938.902} C_VEL
LIN {X 0,Y 425.259,Z 378.136,A -85,B 0,C 180,E1 -9941.956,E2 -9941.956} C_VEL
LIN {X 0,Y 425.279,Z 378.138,A -85,B 0,C 180,E1 -9945.284,E2 -9945.284} C_VEL
LIN {X 0,Y 425.247,Z 378.141,A -85,B 0,C 180,E1 -9948.62,E2 -9948.62} C_VEL
LIN {X 0,Y 425.279,Z 378.137,A -85,B 0,C 180,E1 -9951.101,E2 -9951.101} C_VEL
LIN {X 0,Y 425.313,Z 378.128,A -85,B 0,C 180,E1 -9954.252,E2 -9954.252} C_VEL
LIN {X 0,Y 426.312,Z 380.974,A -85,B 0,C 180,E1 -9954.396,E2 -9954.396} C_VEL
LIN {X 0,Y 435.247,Z 397.843,A -85,B 0,C 180,E1 -9955.391,E2 -9955.391} C_VEL
LIN {X 0,Y 438.219,Z 404.036,A -85,B 0,C 180,E1 -9955.72,E2 -9955.72} C_VEL
LIN {X 0,Y 436.577,Z 504.81,A -85,B 0,C 180,E1 -9957.452,E2 -9957.452} C_VEL
LIN {X 0,Y 436.333,Z 520.322,A -85,B 0,C 180,E1 -9957.858,E2 -9957.858} C_VEL
LIN {X 0,Y 435.88,Z 534.337,A -85,B 0,C 180,E1 -9958.4,E2 -9958.4} C_VEL
LIN {X 0,Y 435.118,Z 548.915,A -85,B 0,C 180,E1 -9959.154,E2 -9959.154} C_VEL
LIN {X 0,Y 434.291,Z 562.074,A -85,B 0,C 180,E1 -9960.025,E2 -9960.025} C_VEL
LIN {X 0,Y 433.283,Z 574.539,A -85,B 0,C 180,E1 -9961.037,E2 -9961.037} C_VEL
LIN {X 0,Y 432.114,Z 586.891,A -85,B 0,C 180,E1 -9962.254,E2 -9962.254} C_VEL
LIN {X 0,Y 430.965,Z 598.522,A -85,B 0,C 180,E1 -9963.644,E2 -9963.644} C_VEL
LIN {X 0,Y 429.866,Z 608.721,A -85,B 0,C 180,E1 -9965.104,E2 -9965.104} C_VEL
LIN {X 0,Y 428.783,Z 617.632,A -85,B 0,C 180,E1 -9966.618,E2 -9966.618} C_VEL
LIN {X 0,Y 427.835,Z 625.923,A -85,B 0,C 180,E1 -9968.31,E2 -9968.31} C_VEL
LIN {X 0,Y 427.159,Z 632.007,A -85,B 0,C 180,E1 -9969.788,E2 -9969.788} C_VEL
LIN {X 0,Y 426.438,Z 638.587,A -85,B 0,C 180,E1 -9971.753,E2 -9971.753} C_VEL
LIN {X 0,Y 425.993,Z 642.459,A -85,B 0,C 180,E1 -9973.2,E2 -9973.2} C_VEL
LIN {X 0,Y 425.127,Z 644.322,A -85,B 0,C 180,E1 -9973.948,E2 -9973.948} C_VEL
LIN {X 0,Y 422.014,Z 647.184,A -85,B 0,C 180,E1 -9975.161,E2 -9975.161} C_VEL
LIN {X 0,Y 419.467,Z 649.13,A -85,B 0,C 180,E1 -9976.152,E2 -9976.152} C_VEL
LIN {X 0,Y 418.37,Z 650.286,A -85,B 0,C 180,E1 -9976.932,E2 -9976.932} C_VEL
LIN {X 0,Y 418.275,Z 650.576,A -85,B 0,C 180,E1 -9977.198,E2 -9977.198} C_VEL
LIN {X 0,Y 418.104,Z 652.158,A -85,B 0,C 180,E1 -9979.345,E2 -9979.345} C_VEL
LIN {X 0,Y 418.079,Z 652.418,A -85,B 0,C 180,E1 -9981.299,E2 -9981.299} C_VEL
LIN {X 0,Y 418.187,Z 651.576,A -85,B 0,C 180,E1 -9983.245,E2 -9983.245} C_VEL
LIN {X 0,Y 418.204,Z 649.662,A -85,B 0,C 180,E1 -9985.18,E2 -9985.18} C_VEL
LIN {X 0,Y 418.52,Z 646.531,A -85,B 0,C 180,E1 -9987.113,E2 -9987.113} C_VEL
LIN {X 0,Y 418.759,Z 642.231,A -85,B 0,C 180,E1 -9989.039,E2 -9989.039} C_VEL
LIN {X 0,Y 419.381,Z 636.593,A -85,B 0,C 180,E1 -9990.961,E2 -9990.961} C_VEL
LIN {X 0,Y 420.102,Z 629.513,A -85,B 0,C 180,E1 -9992.877,E2 -9992.877} C_VEL
LIN {X 0,Y 420.874,Z 621.941,A -85,B 0,C 180,E1 -9994.55,E2 -9994.55} C_VEL
LIN {X 0,Y 421.841,Z 612.853,A -85,B 0,C 180,E1 -9996.217,E2 -9996.217} C_VEL
LIN {X 0,Y 422.927,Z 601.908,A -85,B 0,C 180,E1 -9997.88,E2 -9997.88} C_VEL
LIN {X 0,Y 423.968,Z 590.619,A -85,B 0,C 180,E1 -9999.301,E2 -9999.301} C_VEL
LIN {X 0,Y 424.837,Z 579.448,A -85,B 0,C 180,E1 -10000.485,E2 -10000.485} C_VEL
LIN {X 0,Y 425.869,Z 567.399,A -85,B 0,C 180,E1 -10001.543,E2 -10001.543} C_VEL
LIN {X 0,Y 426.748,Z 554.394,A -85,B 0,C 180,E1 -10002.483,E2 -10002.483} C_VEL
LIN {X 0,Y 427.533,Z 540.015,A -85,B 0,C 180,E1 -10003.305,E2 -10003.305} C_VEL
LIN {X 0,Y 428.076,Z 524.604,A -85,B 0,C 180,E1 -10003.969,E2 -10003.969} C_VEL
LIN {X 0,Y 428.36,Z 509.123,A -85,B 0,C 180,E1 -10004.429,E2 -10004.429} C_VEL
LIN {X 0,Y 429.248,Z 440.348,A -85,B 0,C 180,E1 -10005.629,E2 -10005.629} C_VEL
LIN {X 0,Y 429.728,Z 404.59,A -85,B 0,C 180,E1 -10006.242,E2 -10006.242} C_VEL
LIN {X 0,Y 419.025,Z 381.493,A -85,B 0,C 180,E1 -10007.317,E2 -10007.317} C_VEL
LIN {X 0,Y 418.239,Z 379.028,A -85,B 0,C 180,E1 -10007.412,E2 -10007.412} C_VEL
LIN {X 0,Y 418.239,Z 379.013,A -85,B 0,C 180,E1 -10010.663,E2 -10010.663} C_VEL
LIN {X 0,Y 418.224,Z 379.014,A -85,B 0,C 180,E1 -10013.785,E2 -10013.785} C_VEL
LIN {X 0,Y 418.198,Z 379.02,A -85,B 0,C 180,E1 -10017.04,E2 -10017.04} C_VEL
LIN {X 0,Y 418.233,Z 378.998,A -85,B 0,C 180,E1 -10020.273,E2 -10020.273} C_VEL
LIN {X 0,Y 418.226,Z 379.011,A -85,B 0,C 180,E1 -10023.679,E2 -10023.679} C_VEL
LIN {X 0,Y 418.23,Z 379.013,A -85,B 0,C 180,E1 -10027.224,E2 -10027.224} C_VEL
LIN {X 0,Y 418.204,Z 379.013,A -85,B 0,C 180,E1 -10030.866,E2 -10030.866} C_VEL
LIN {X 0,Y 418.177,Z 379.016,A -85,B 0,C 180,E1 -10033.724,E2 -10033.724} C_VEL
LIN {X 0,Y 418.194,Z 379.015,A -85,B 0,C 180,E1 -10036.446,E2 -10036.446} C_VEL
LIN {X 0,Y 418.203,Z 379.018,A -85,B 0,C 180,E1 -10039.132,E2 -10039.132} C_VEL
LIN {X 0,Y 418.229,Z 379.01,A -85,B 0,C 180,E1 -10042.774,E2 -10042.774} C_VEL
LIN {X 0,Y 418.222,Z 379.006,A -85,B 0,C 180,E1 -10046.32,E2 -10046.32} C_VEL
LIN {X 0,Y 418.227,Z 379.011,A -85,B 0,C 180,E1 -10049.726,E2 -10049.726} C_VEL
LIN {X 0,Y 418.194,Z 379.018,A -85,B 0,C 180,E1 -10053.015,E2 -10053.015} C_VEL
LIN {X 0,Y 418.248,Z 379.003,A -85,B 0,C 180,E1 -10056.216,E2 -10056.216} C_VEL
LIN {X 0,Y 418.242,Z 379.014,A -85,B 0,C 180,E1 -10059.336,E2 -10059.336} C_VEL
LIN {X 0,Y 418.27,Z 379.003,A -85,B 0,C 180,E1 -10062.395,E2 -10062.395} C_VEL
LIN {X 0,Y 418.285,Z 379.004,A -85,B 0,C 180,E1 -10065.402,E2 -10065.402} C_VEL
LIN {X 0,Y 418.301,Z 378.977,A -85,B 0,C 180,E1 -10068.368,E2 -10068.368} C_VEL
LIN {X 0,Y 418.438,Z 378.979,A -85,B 0,C 180,E1 -10072.278,E2 -10072.278} C_VEL
LIN {X 0,Y 418.459,Z 378.982,A -85,B 0,C 180,E1 -10074.216,E2 -10074.216} C_VEL
LIN {X 0,Y 418.519,Z 378.969,A -85,B 0,C 180,E1 -10078.075,E2 -10078.075} C_VEL
LIN {X 0,Y 418.526,Z 378.973,A -85,B 0,C 180,E1 -10081.924,E2 -10081.924} C_VEL
LIN {X 0,Y 418.455,Z 378.986,A -85,B 0,C 180,E1 -10085.783,E2 -10085.783} C_VEL
LIN {X 0,Y 418.359,Z 378.989,A -85,B 0,C 180,E1 -10088.696,E2 -10088.696} C_VEL
LIN {X 0,Y 418.301,Z 379.007,A -85,B 0,C 180,E1 -10091.631,E2 -10091.631} C_VEL
LIN {X 0,Y 418.254,Z 379.002,A -85,B 0,C 180,E1 -10094.598,E2 -10094.598} C_VEL
LIN {X 0,Y 418.227,Z 379.015,A -85,B 0,C 180,E1 -10097.606,E2 -10097.606} C_VEL
LIN {X 0,Y 418.227,Z 379.011,A -85,B 0,C 180,E1 -10100.664,E2 -10100.664} C_VEL
LIN {X 0,Y 418.245,Z 379.012,A -85,B 0,C 180,E1 -10103.783,E2 -10103.783} C_VEL
LIN {X 0,Y 418.199,Z 379.012,A -85,B 0,C 180,E1 -10107.043,E2 -10107.043} C_VEL
LIN {X 0,Y 418.231,Z 379.013,A -85,B 0,C 180,E1 -10110.273,E2 -10110.273} C_VEL
LIN {X 0,Y 418.224,Z 379.006,A -85,B 0,C 180,E1 -10113.679,E2 -10113.679} C_VEL
LIN {X 0,Y 418.225,Z 379.015,A -85,B 0,C 180,E1 -10117.225,E2 -10117.225} C_VEL
LIN {X 0,Y 418.2,Z 379.015,A -85,B 0,C 180,E1 -10120.867,E2 -10120.867} C_VEL
LIN {X 0,Y 418.196,Z 379.018,A -85,B 0,C 180,E1 -10123.728,E2 -10123.728} C_VEL
LIN {X 0,Y 418.194,Z 379.02,A -85,B 0,C 180,E1 -10126.448,E2 -10126.448} C_VEL
LIN {X 0,Y 418.2,Z 378.998,A -85,B 0,C 180,E1 -10129.134,E2 -10129.134} C_VEL
LIN {X 0,Y 418.251,Z 379.011,A -85,B 0,C 180,E1 -10132.811,E2 -10132.811} C_VEL
LIN {X 0,Y 423.443,Z 398.173,A -85,B 0,C 180,E1 -10135.814,E2 -10135.814} C_VEL
LIN {X 0,Y 426.189,Z 409.896,A -85,B 0,C 180,E1 -10137.544,E2 -10137.544} C_VEL
LIN {X 0,Y 424.771,Z 430.022,A -85,B 0,C 180,E1 -10140.104,E2 -10140.104} C_VEL
LIN {X 0,Y 423.324,Z 452.732,A -85,B 0,C 180,E1 -10142.969,E2 -10142.969} C_VEL
LIN {X 0,Y 423.175,Z 454.779,A -85,B 0,C 180,E1 -10143.225,E2 -10143.225} C_VEL
LIN {X 0,Y 429.205,Z 498.641,A -85,B 0,C 180,E1 -10144.359,E2 -10144.359} C_VEL
LIN {X 0,Y 427.321,Z 619.11,A -85,B 0,C 180,E1 -10146.399,E2 -10146.399} C_VEL
LIN {X 0,Y 426.836,Z 633.804,A -85,B 0,C 180,E1 -10146.756,E2 -10146.756} C_VEL
LIN {X 0,Y 425.881,Z 649.178,A -85,B 0,C 180,E1 -10147.311,E2 -10147.311} C_VEL
LIN {X 0,Y 424.728,Z 664.042,A -85,B 0,C 180,E1 -10148.045,E2 -10148.045} C_VEL
LIN {X 0,Y 423.549,Z 678.498,A -85,B 0,C 180,E1 -10148.972,E2 -10148.972} C_VEL
LIN {X 0,Y 422.361,Z 692.055,A -85,B 0,C 180,E1 -10150.055,E2 -10150.055} C_VEL
LIN {X 0,Y 421.234,Z 704.559,A -85,B 0,C 180,E1 -10151.266,E2 -10151.266} C_VEL
LIN {X 0,Y 420.071,Z 717.053,A -85,B 0,C 180,E1 -10152.725,E2 -10152.725} C_VEL
LIN {X 0,Y 419.187,Z 727.585,A -85,B 0,C 180,E1 -10154.19,E2 -10154.19} C_VEL
LIN {X 0,Y 418.439,Z 737.894,A -85,B 0,C 180,E1 -10155.905,E2 -10155.905} C_VEL
LIN {X 0,Y 417.847,Z 747.574,A -85,B 0,C 180,E1 -10157.863,E2 -10157.863} C_VEL
LIN {X 0,Y 417.604,Z 755.43,A -85,B 0,C 180,E1 -10159.822,E2 -10159.822} C_VEL
LIN {X 0,Y 417.532,Z 761.683,A -85,B 0,C 180,E1 -10161.774,E2 -10161.774} C_VEL
LIN {X 0,Y 417.584,Z 766.109,A -85,B 0,C 180,E1 -10163.544,E2 -10163.544} C_VEL
LIN {X 0,Y 417.662,Z 769.176,A -85,B 0,C 180,E1 -10165.173,E2 -10165.173} C_VEL
LIN {X 0,Y 417.695,Z 771.668,A -85,B 0,C 180,E1 -10167.106,E2 -10167.106} C_VEL
LIN {X 0,Y 417.894,Z 772.956,A -85,B 0,C 180,E1 -10169.036,E2 -10169.036} C_VEL
LIN {X 0,Y 417.895,Z 772.956,A -85,B 0,C 180,E1 -10170.963,E2 -10170.963} C_VEL
LIN {X 0,Y 417.688,Z 771.728,A -85,B 0,C 180,E1 -10172.893,E2 -10172.893} C_VEL
LIN {X 0,Y 417.676,Z 769.322,A -85,B 0,C 180,E1 -10174.826,E2 -10174.826} C_VEL
LIN {X 0,Y 417.601,Z 765.543,A -85,B 0,C 180,E1 -10176.814,E2 -10176.814} C_VEL
LIN {X 0,Y 417.49,Z 760.653,A -85,B 0,C 180,E1 -10178.714,E2 -10178.714} C_VEL
LIN {X 0,Y 417.648,Z 754.22,A -85,B 0,C 180,E1 -10180.666,E2 -10180.666} C_VEL
LIN {X 0,Y 417.919,Z 746.188,A -85,B 0,C 180,E1 -10182.627,E2 -10182.627} C_VEL
LIN {X 0,Y 418.528,Z 737.685,A -85,B 0,C 180,E1 -10184.34,E2 -10184.34} C_VEL
LIN {X 0,Y 419.358,Z 727.547,A -85,B 0,C 180,E1 -10186.052,E2 -10186.052} C_VEL
LIN {X 0,Y 420.412,Z 716.142,A -85,B 0,C 180,E1 -10187.662,E2 -10187.662} C_VEL
LIN {X 0,Y 421.625,Z 703.99,A -85,B 0,C 180,E1 -10189.093,E2 -10189.093} C_VEL
LIN {X 0,Y 422.977,Z 690.4,A -85,B 0,C 180,E1 -10190.421,E2 -10190.421} C_VEL
LIN {X 0,Y 424.42,Z 676.994,A -85,B 0,C 180,E1 -10191.482,E2 -10191.482} C_VEL
LIN {X 0,Y 425.662,Z 662.83,A -85,B 0,C 180,E1 -10192.392,E2 -10192.392} C_VEL
LIN {X 0,Y 426.989,Z 647.941,A -85,B 0,C 180,E1 -10193.126,E2 -10193.126} C_VEL
LIN {X 0,Y 428.061,Z 632.362,A -85,B 0,C 180,E1 -10193.686,E2 -10193.686} C_VEL
LIN {X 0,Y 428.706,Z 617.759,A -85,B 0,C 180,E1 -10194.033,E2 -10194.033} C_VEL
LIN {X 0,Y 430.775,Z 499.467,A -85,B 0,C 180,E1 -10196.073,E2 -10196.073} C_VEL
LIN {X 0,Y 427.026,Z 471.16,A -85,B 0,C 180,E1 -10196.865,E2 -10196.865} C_VEL
LIN {X 0,Y 424.074,Z 453.245,A -85,B 0,C 180,E1 -10197.44,E2 -10197.44} C_VEL
LIN {X 0,Y 426.091,Z 427.819,A -85,B 0,C 180,E1 -10200.75,E2 -10200.75} C_VEL
LIN {X 0,Y 427.46,Z 411.868,A -85,B 0,C 180,E1 -10202.857,E2 -10202.857} C_VEL
LIN {X 0,Y 423.76,Z 397.116,A -85,B 0,C 180,E1 -10205.235,E2 -10205.235} C_VEL
LIN {X 0,Y 418.968,Z 381.551,A -85,B 0,C 180,E1 -10207.964,E2 -10207.964} C_VEL
LIN {X 0,Y 418.24,Z 379.013,A -85,B 0,C 180,E1 -10208.442,E2 -10208.442} C_VEL
LIN {X 0,Y 418.211,Z 379.015,A -85,B 0,C 180,E1 -10212.235,E2 -10212.235} C_VEL
